    movel([0.094218, -1.402546, -2.554876, -0.754968, 1.570796, 1.665014],accel_mss,speed_ms,0,blend_radius_m)
    movel([0.093145, -1.402897, -2.554616, -0.754876, 1.570796, 1.663941],accel_mss,speed_ms,0,blend_radius_m)
    movel([0.092652, -1.403004, -2.554537, -0.754848, 1.570796, 1.663448],accel_mss,speed_ms,0,blend_radius_m)
    movel([0.092424, -1.402949, -2.554578, -0.754862, 1.570796, 1.663220],accel_mss,speed_ms,0,blend_radius_m)
    movel([0.092353, -1.402753, -2.554722, -0.754913, 1.570796, 1.663149],accel_mss,speed_ms,0,blend_radius_m)
    movel([0.092529, -1.402431, -2.554960, -0.754998, 1.570796, 1.663326],accel_mss,speed_ms,0,blend_radius_m)
    movel([0.093124, -1.402001, -2.555277, -0.755111, 1.570796, 1.663921],accel_mss,speed_ms,0,blend_radius_m)
    movel([0.094351, -1.401555, -2.555606, -0.755228, 1.570796, 1.665147],accel_mss,speed_ms,0,blend_radius_m)
    movel([0.095795, -1.401115, -2.555930, -0.755344, 1.570796, 1.666591],accel_mss,speed_ms,0,blend_radius_m)
    speed_ms = 0.003
    movel([0.095795, -1.404350, -2.557382, -0.750656, 1.570796, 1.666591],accel_mss,speed_ms,0,blend_radius_m)
    speed_ms = 0.007
    movel([0.097270, -1.403994, -2.557646, -0.750749, 1.570796, 1.668067],accel_mss,speed_ms,0,blend_radius_m)
    movel([0.098200, -1.403807, -2.557784, -0.750798, 1.570796, 1.668996],accel_mss,speed_ms,0,blend_radius_m)
    movel([0.098654, -1.403741, -2.557833, -0.750815, 1.570796, 1.669451],accel_mss,speed_ms,0,blend_radius_m)
    movel([0.098932, -1.403749, -2.557827, -0.750813, 1.570796, 1.669729],accel_mss,speed_ms,0,blend_radius_m)
    movel([0.099151, -1.403824, -2.557771, -0.750794, 1.570796, 1.669947],accel_mss,speed_ms,0,blend_radius_m)
    movel([0.099338, -1.403962, -2.557669, -0.750758, 1.570796, 1.670134],accel_mss,speed_ms,0,blend_radius_m)
    movel([0.099360, -1.404241, -2.557463, -0.750685, 1.570796, 1.670156],accel_mss,speed_ms,0,blend_radius_m)
    movel([0.099047, -1.404511, -2.557263, -0.750614, 1.570796, 1.669844],accel_mss,speed_ms,0,blend_radius_m)
    movel([0.098716, -1.404617, -2.557185, -0.750587, 1.570796, 1.669513],accel_mss,speed_ms,0,blend_radius_m)
    movel([0.098213, -1.404743, -2.557092, -0.750554, 1.570796, 1.669009],accel_mss,speed_ms,0,blend_radius_m)
    movel([0.097407, -1.404912, -2.556967, -0.750510, 1.570796, 1.668203],accel_mss,speed_ms,0,blend_radius_m)
    movel([0.096581, -1.405094, -2.556832, -0.750463, 1.570796, 1.667377],accel_mss,speed_ms,0,blend_radius_m)
    movel([0.095800, -1.405291, -2.556686, -0.750412, 1.570796, 1.666597],accel_mss,speed_ms,0,blend_radius_m)
    movel([0.095027, -1.405514, -2.556521, -0.750354, 1.570796, 1.665823],accel_mss,speed_ms,0,blend_radius_m)
    movel([0.094218, -1.405777, -2.556325, -0.750286, 1.570796, 1.665014],accel_mss,speed_ms,0,blend_radius_m)
    movel([0.093145, -1.406127, -2.556066, -0.750196, 1.570796, 1.663941],accel_mss,speed_ms,0,blend_radius_m)
    movel([0.092652, -1.406234, -2.555986, -0.750168, 1.570796, 1.663448],accel_mss,speed_ms,0,blend_radius_m)
    movel([0.092424, -1.406179, -2.556027, -0.750182, 1.570796, 1.663220],accel_mss,speed_ms,0,blend_radius_m)
    movel([0.092353, -1.405984, -2.556172, -0.750233, 1.570796, 1.663149],accel_mss,speed_ms,0,blend_radius_m)
    movel([0.092529, -1.405663, -2.556410, -0.750316, 1.570796, 1.663326],accel_mss,speed_ms,0,blend_radius_m)
    movel([0.093124, -1.405234, -2.556728, -0.750427, 1.570796, 1.663921],accel_mss,speed_ms,0,blend_radius_m)
    movel([0.094351, -1.404789, -2.557058, -0.750542, 1.570796, 1.665147],accel_mss,speed_ms,0,blend_radius_m)
    movel([0.095795, -1.404350, -2.557382, -0.750656, 1.570796, 1.666591],accel_mss,speed_ms,0,blend_radius_m)
    speed_ms = 0.003
    movel([0.095795, -1.391535, -2.551523, -0.769331, 1.570796, 1.666591],accel_mss,speed_ms,0,blend_radius_m)
    speed_ms = 1.000
    movel([0.095795, -1.366921, -2.539410, -0.806058, 1.570796, 1.666591],accel_mss,speed_ms,0,blend_radius_m)
    movel([0.095058, -1.368794, -2.538098, -0.805497, 1.570796, 1.665854],accel_mss,speed_ms,0,blend_radius_m)
    movel([0.095058, -1.393374, -2.550187, -0.768828, 1.570796, 1.665854],accel_mss,speed_ms,0,blend_radius_m)
    speed_ms = 0.003
    movel([0.095058, -1.402939, -2.554585, -0.754865, 1.570796, 1.665854],accel_mss,speed_ms,0,blend_radius_m)
    speed_ms = 0.007
    movel([0.096957, -1.402395, -2.554986, -0.755007, 1.570796, 1.667754],accel_mss,speed_ms,0,blend_radius_m)
    movel([0.098037, -1.402157, -2.555162, -0.755070, 1.570796, 1.668833],accel_mss,speed_ms,0,blend_radius_m)
    movel([0.098676, -1.402118, -2.555191, -0.755080, 1.570796, 1.669473],accel_mss,speed_ms,0,blend_radius_m)
    movel([0.099066, -1.402259, -2.555087, -0.755043, 1.570796, 1.669862],accel_mss,speed_ms,0,blend_radius_m)
    movel([0.099131, -1.402534, -2.554884, -0.754971, 1.570796, 1.669927],accel_mss,speed_ms,0,blend_radius_m)
    movel([0.098905, -1.402879, -2.554629, -0.754881, 1.570796, 1.669701],accel_mss,speed_ms,0,blend_radius_m)
    movel([0.098649, -1.402995, -2.554544, -0.754850, 1.570796, 1.669445],accel_mss,speed_ms,0,blend_radius_m)
    movel([0.098218, -1.403073, -2.554486, -0.754830, 1.570796, 1.669014],accel_mss,speed_ms,0,blend_radius_m)
    movel([0.097382, -1.403224, -2.554375, -0.754791, 1.570796, 1.668179],accel_mss,speed_ms,0,blend_radius_m)
    movel([0.095577, -1.403702, -2.554021, -0.754666, 1.570796, 1.666373],accel_mss,speed_ms,0,blend_radius_m)
    movel([0.093763, -1.404215, -2.553642, -0.754533, 1.570796, 1.664560],accel_mss,speed_ms,0,blend_radius_m)
    movel([0.092999, -1.404503, -2.553428, -0.754458, 1.570796, 1.663795],accel_mss,speed_ms,0,blend_radius_m)
    movel([0.092709, -1.404629, -2.553335, -0.754425, 1.570796, 1.663506],accel_mss,speed_ms,0,blend_radius_m)
    movel([0.092398, -1.404692, -2.553288, -0.754409, 1.570796, 1.663195],accel_mss,speed_ms,0,blend_radius_m)
    movel([0.092200, -1.404501, -2.553429, -0.754458, 1.570796, 1.662996],accel_mss,speed_ms,0,blend_radius_m)
    movel([0.092240, -1.404260, -2.553608, -0.754521, 1.570796, 1.663036],accel_mss,speed_ms,0,blend_radius_m)
    movel([0.092394, -1.403991, -2.553808, -0.754591, 1.570796, 1.663190],accel_mss,speed_ms,0,blend_radius_m)
    movel([0.092628, -1.403768, -2.553972, -0.754649, 1.570796, 1.663424],accel_mss,speed_ms,0,blend_radius_m)
    movel([0.093075, -1.403542, -2.554139, -0.754707, 1.570796, 1.663871],accel_mss,speed_ms,0,blend_radius_m)
    movel([0.095058, -1.402939, -2.554585, -0.754865, 1.570796, 1.665854],accel_mss,speed_ms,0,blend_radius_m)
    speed_ms = 0.003
    movel([0.095058, -1.406170, -2.556034, -0.750185, 1.570796, 1.665854],accel_mss,speed_ms,0,blend_radius_m)
    speed_ms = 0.007
    movel([0.096957, -1.405627, -2.556437, -0.750325, 1.570796, 1.667754],accel_mss,speed_ms,0,blend_radius_m)
    movel([0.098037, -1.405390, -2.556613, -0.750386, 1.570796, 1.668833],accel_mss,speed_ms,0,blend_radius_m)
    movel([0.098676, -1.405351, -2.556641, -0.750396, 1.570796, 1.669473],accel_mss,speed_ms,0,blend_radius_m)
    movel([0.099066, -1.405491, -2.556537, -0.750360, 1.570796, 1.669862],accel_mss,speed_ms,0,blend_radius_m)
    movel([0.099131, -1.405766, -2.556334, -0.750289, 1.570796, 1.669927],accel_mss,speed_ms,0,blend_radius_m)
    movel([0.098905, -1.406110, -2.556079, -0.750200, 1.570796, 1.669701],accel_mss,speed_ms,0,blend_radius_m)
    movel([0.098649, -1.406225, -2.555993, -0.750171, 1.570796, 1.669445],accel_mss,speed_ms,0,blend_radius_m)
    movel([0.098218, -1.406303, -2.555935, -0.750151, 1.570796, 1.669014],accel_mss,speed_ms,0,blend_radius_m)
    movel([0.097382, -1.406453, -2.555824, -0.750112, 1.570796, 1.668179],accel_mss,speed_ms,0,blend_radius_m)
    movel([0.095577, -1.406930, -2.555469, -0.749989, 1.570796, 1.666373],accel_mss,speed_ms,0,blend_radius_m)
    movel([0.093763, -1.407442, -2.555089, -0.749858, 1.570796, 1.664560],accel_mss,speed_ms,0,blend_radius_m)
    movel([0.092999, -1.407729, -2.554875, -0.749785, 1.570796, 1.663795],accel_mss,speed_ms,0,blend_radius_m)
    movel([0.092709, -1.407855, -2.554782, -0.749753, 1.570796, 1.663506],accel_mss,speed_ms,0,blend_radius_m)
    movel([0.092398, -1.407917, -2.554735, -0.749737, 1.570796, 1.663195],accel_mss,speed_ms,0,blend_radius_m)
    movel([0.092200, -1.407728, -2.554876, -0.749785, 1.570796, 1.662996],accel_mss,speed_ms,0,blend_radius_m)
    movel([0.092240, -1.407487, -2.555056, -0.749847, 1.570796, 1.663036],accel_mss,speed_ms,0,blend_radius_m)
    movel([0.092394, -1.407218, -2.555255, -0.749916, 1.570796, 1.663190],accel_mss,speed_ms,0,blend_radius_m)
    movel([0.092628, -1.406997, -2.555420, -0.749972, 1.570796, 1.663424],accel_mss,speed_ms,0,blend_radius_m)
    movel([0.093075, -1.406771, -2.555588, -0.750030, 1.570796, 1.663871],accel_mss,speed_ms,0,blend_radius_m)
    movel([0.095058, -1.406170, -2.556034, -0.750185, 1.570796, 1.665854],accel_mss,speed_ms,0,blend_radius_m)
    speed_ms = 0.003
    movel([0.095058, -1.393374, -2.550187, -0.768828, 1.570796, 1.665854],accel_mss,speed_ms,0,blend_radius_m)
    speed_ms = 1.000
    movel([0.095058, -1.368794, -2.538098, -0.805497, 1.570796, 1.665854],accel_mss,speed_ms,0,blend_radius_m)
    movel([0.095035, -1.370360, -2.536997, -0.805032, 1.570796, 1.665831],accel_mss,speed_ms,0,blend_radius_m)
    movel([0.095035, -1.394911, -2.549067, -0.768411, 1.570796, 1.665831],accel_mss,speed_ms,0,blend_radius_m)
    speed_ms = 0.003
    movel([0.095035, -1.404463, -2.553458, -0.754468, 1.570796, 1.665831],accel_mss,speed_ms,0,blend_radius_m)
    speed_ms = 0.007
    movel([0.096678, -1.404013, -2.553791, -0.754585, 1.570796, 1.667474],accel_mss,speed_ms,0,blend_radius_m)
    movel([0.097776, -1.403780, -2.553963, -0.754646, 1.570796, 1.668573],accel_mss,speed_ms,0,blend_radius_m)
    movel([0.098503, -1.403710, -2.554016, -0.754664, 1.570796, 1.669299],accel_mss,speed_ms,0,blend_radius_m)
    movel([0.098867, -1.403822, -2.553932, -0.754635, 1.570796, 1.669663],accel_mss,speed_ms,0,blend_radius_m)
    movel([0.098943, -1.404146, -2.553692, -0.754550, 1.570796, 1.669739],accel_mss,speed_ms,0,blend_radius_m)
    movel([0.098660, -1.404518, -2.553417, -0.754454, 1.570796, 1.669456],accel_mss,speed_ms,0,blend_radius_m)
    movel([0.098382, -1.404581, -2.553370, -0.754438, 1.570796, 1.669178],accel_mss,speed_ms,0,blend_radius_m)
    movel([0.098132, -1.404608, -2.553350, -0.754431, 1.570796, 1.668928],accel_mss,speed_ms,0,blend_radius_m)
    movel([0.097854, -1.404624, -2.553339, -0.754426, 1.570796, 1.668651],accel_mss,speed_ms,0,blend_radius_m)
    movel([0.096922, -1.404748, -2.553246, -0.754394, 1.570796, 1.667719],accel_mss,speed_ms,0,blend_radius_m)
    movel([0.095411, -1.405123, -2.552968, -0.754297, 1.570796, 1.666208],accel_mss,speed_ms,0,blend_radius_m)
    movel([0.093895, -1.405570, -2.552637, -0.754182, 1.570796, 1.664692],accel_mss,speed_ms,0,blend_radius_m)
    movel([0.092949, -1.405958, -2.552349, -0.754082, 1.570796, 1.663745],accel_mss,speed_ms,0,blend_radius_m)
    movel([0.092619, -1.406115, -2.552232, -0.754042, 1.570796, 1.663415],accel_mss,speed_ms,0,blend_radius_m)
    movel([0.092226, -1.406242, -2.552137, -0.754009, 1.570796, 1.663023],accel_mss,speed_ms,0,blend_radius_m)
    movel([0.092027, -1.406107, -2.552238, -0.754044, 1.570796, 1.662823],accel_mss,speed_ms,0,blend_radius_m)
    movel([0.092203, -1.405669, -2.552563, -0.754157, 1.570796, 1.663000],accel_mss,speed_ms,0,blend_radius_m)
    movel([0.092457, -1.405414, -2.552753, -0.754222, 1.570796, 1.663253],accel_mss,speed_ms,0,blend_radius_m)
    movel([0.092744, -1.405218, -2.552898, -0.754273, 1.570796, 1.663541],accel_mss,speed_ms,0,blend_radius_m)
    movel([0.093114, -1.405050, -2.553023, -0.754316, 1.570796, 1.663910],accel_mss,speed_ms,0,blend_radius_m)
    movel([0.093718, -1.404848, -2.553172, -0.754368, 1.570796, 1.664514],accel_mss,speed_ms,0,blend_radius_m)
    movel([0.095035, -1.404463, -2.553458, -0.754468, 1.570796, 1.665831],accel_mss,speed_ms,0,blend_radius_m)
    speed_ms = 0.003
    movel([0.095035, -1.407689, -2.554905, -0.749795, 1.570796, 1.665831],accel_mss,speed_ms,0,blend_radius_m)
    speed_ms = 0.007
    movel([0.096678, -1.407240, -2.555239, -0.749910, 1.570796, 1.667474],accel_mss,speed_ms,0,blend_radius_m)
    movel([0.097776, -1.407008, -2.555411, -0.749969, 1.570796, 1.668573],accel_mss,speed_ms,0,blend_radius_m)
    movel([0.098503, -1.406938, -2.555464, -0.749987, 1.570796, 1.669299],accel_mss,speed_ms,0,blend_radius_m)
    movel([0.098867, -1.407050, -2.555380, -0.749959, 1.570796, 1.669663],accel_mss,speed_ms,0,blend_radius_m)
    movel([0.098943, -1.407374, -2.555140, -0.749876, 1.570796, 1.669739],accel_mss,speed_ms,0,blend_radius_m)
    movel([0.098660, -1.407744, -2.554864, -0.749781, 1.570796, 1.669456],accel_mss,speed_ms,0,blend_radius_m)
    movel([0.098382, -1.407807, -2.554817, -0.749765, 1.570796, 1.669178],accel_mss,speed_ms,0,blend_radius_m)
    movel([0.098132, -1.407834, -2.554797, -0.749758, 1.570796, 1.668928],accel_mss,speed_ms,0,blend_radius_m)
    movel([0.097854, -1.407850, -2.554785, -0.749754, 1.570796, 1.668651],accel_mss,speed_ms,0,blend_radius_m)
    movel([0.096922, -1.407974, -2.554693, -0.749722, 1.570796, 1.667719],accel_mss,speed_ms,0,blend_radius_m)
    movel([0.095411, -1.408348, -2.554414, -0.749627, 1.570796, 1.666208],accel_mss,speed_ms,0,blend_radius_m)
    movel([0.093895, -1.408794, -2.554082, -0.749514, 1.570796, 1.664692],accel_mss,speed_ms,0,blend_radius_m)
    movel([0.092949, -1.409180, -2.553793, -0.749416, 1.570796, 1.663745],accel_mss,speed_ms,0,blend_radius_m)
    movel([0.092619, -1.409336, -2.553676, -0.749376, 1.570796, 1.663415],accel_mss,speed_ms,0,blend_radius_m)
    movel([0.092226, -1.409464, -2.553581, -0.749344, 1.570796, 1.663023],accel_mss,speed_ms,0,blend_radius_m)
    movel([0.092027, -1.409329, -2.553682, -0.749378, 1.570796, 1.662823],accel_mss,speed_ms,0,blend_radius_m)
    movel([0.092203, -1.408892, -2.554008, -0.749489, 1.570796, 1.663000],accel_mss,speed_ms,0,blend_radius_m)
    movel([0.092457, -1.408637, -2.554198, -0.749553, 1.570796, 1.663253],accel_mss,speed_ms,0,blend_radius_m)
    movel([0.092744, -1.408442, -2.554344, -0.749603, 1.570796, 1.663541],accel_mss,speed_ms,0,blend_radius_m)
    movel([0.093114, -1.408275, -2.554469, -0.749646, 1.570796, 1.663910],accel_mss,speed_ms,0,blend_radius_m)
    movel([0.093718, -1.408074, -2.554618, -0.749697, 1.570796, 1.664514],accel_mss,speed_ms,0,blend_radius_m)
    movel([0.095035, -1.407689, -2.554905, -0.749795, 1.570796, 1.665831],accel_mss,speed_ms,0,blend_radius_m)
    speed_ms = 0.003
    movel([0.095035, -1.394911, -2.549067, -0.768411, 1.570796, 1.665831],accel_mss,speed_ms,0,blend_radius_m)
    speed_ms = 1.000
    movel([0.095035, -1.370360, -2.536997, -0.805032, 1.570796, 1.665831],accel_mss,speed_ms,0,blend_radius_m)
    movel([0.094639, -1.371914, -2.535902, -0.804573, 1.570796, 1.665435],accel_mss,speed_ms,0,blend_radius_m)
    movel([0.094639, -1.396436, -2.547952, -0.768001, 1.570796, 1.665435],accel_mss,speed_ms,0,blend_radius_m)
    speed_ms = 0.003
    movel([0.094639, -1.405976, -2.552335, -0.754078, 1.570796, 1.665435],accel_mss,speed_ms,0,blend_radius_m)
    speed_ms = 0.007
    movel([0.095700, -1.405698, -2.552542, -0.754149, 1.570796, 1.666496],accel_mss,speed_ms,0,blend_radius_m)
    movel([0.097708, -1.405190, -2.552919, -0.754280, 1.570796, 1.668504],accel_mss,speed_ms,0,blend_radius_m)
    movel([0.098496, -1.405331, -2.552814, -0.754244, 1.570796, 1.669292],accel_mss,speed_ms,0,blend_radius_m)
    movel([0.099084, -1.405493, -2.552694, -0.754202, 1.570796, 1.669880],accel_mss,speed_ms,0,blend_radius_m)
    movel([0.099446, -1.405731, -2.552517, -0.754141, 1.570796, 1.670242],accel_mss,speed_ms,0,blend_radius_m)
    movel([0.099663, -1.406106, -2.552239, -0.754044, 1.570796, 1.670460],accel_mss,speed_ms,0,blend_radius_m)
    movel([0.099786, -1.406703, -2.551795, -0.753891, 1.570796, 1.670583],accel_mss,speed_ms,0,blend_radius_m)
    movel([0.099688, -1.407004, -2.551571, -0.753814, 1.570796, 1.670484],accel_mss,speed_ms,0,blend_radius_m)
    movel([0.099544, -1.407333, -2.551326, -0.753730, 1.570796, 1.670341],accel_mss,speed_ms,0,blend_radius_m)
    movel([0.099344, -1.407622, -2.551110, -0.753657, 1.570796, 1.670140],accel_mss,speed_ms,0,blend_radius_m)
    movel([0.098360, -1.408089, -2.550762, -0.753538, 1.570796, 1.669156],accel_mss,speed_ms,0,blend_radius_m)
    movel([0.096049, -1.408788, -2.550240, -0.753361, 1.570796, 1.666845],accel_mss,speed_ms,0,blend_radius_m)
    movel([0.093670, -1.409447, -2.549747, -0.753195, 1.570796, 1.664466],accel_mss,speed_ms,0,blend_radius_m)
    movel([0.091851, -1.409859, -2.549439, -0.753091, 1.570796, 1.662647],accel_mss,speed_ms,0,blend_radius_m)
    movel([0.091060, -1.409980, -2.549348, -0.753061, 1.570796, 1.661856],accel_mss,speed_ms,0,blend_radius_m)
    movel([0.090671, -1.409936, -2.549381, -0.753072, 1.570796, 1.661467],accel_mss,speed_ms,0,blend_radius_m)
    movel([0.090493, -1.409731, -2.549535, -0.753123, 1.570796, 1.661289],accel_mss,speed_ms,0,blend_radius_m)
    movel([0.090475, -1.409302, -2.549856, -0.753231, 1.570796, 1.661272],accel_mss,speed_ms,0,blend_radius_m)
    movel([0.090698, -1.408553, -2.550415, -0.753420, 1.570796, 1.661494],accel_mss,speed_ms,0,blend_radius_m)
    movel([0.091185, -1.407836, -2.550951, -0.753602, 1.570796, 1.661982],accel_mss,speed_ms,0,blend_radius_m)
    movel([0.091933, -1.407176, -2.551443, -0.753770, 1.570796, 1.662729],accel_mss,speed_ms,0,blend_radius_m)
    movel([0.092913, -1.406594, -2.551876, -0.753919, 1.570796, 1.663709],accel_mss,speed_ms,0,blend_radius_m)
    movel([0.093405, -1.406375, -2.552039, -0.753975, 1.570796, 1.664201],accel_mss,speed_ms,0,blend_radius_m)
    movel([0.093939, -1.406183, -2.552182, -0.754025, 1.570796, 1.664735],accel_mss,speed_ms,0,blend_radius_m)
    movel([0.094639, -1.405976, -2.552335, -0.754078, 1.570796, 1.665435],accel_mss,speed_ms,0,blend_radius_m)
    speed_ms = 0.003
    movel([0.094639, -1.409198, -2.553780, -0.749411, 1.570796, 1.665435],accel_mss,speed_ms,0,blend_radius_m)
    speed_ms = 0.007
    movel([0.095700, -1.408921, -2.553987, -0.749481, 1.570796, 1.666496],accel_mss,speed_ms,0,blend_radius_m)
    movel([0.097708, -1.408414, -2.554365, -0.749610, 1.570796, 1.668504],accel_mss,speed_ms,0,blend_radius_m)
    movel([0.098496, -1.408555, -2.554259, -0.749574, 1.570796, 1.669292],accel_mss,speed_ms,0,blend_radius_m)
    movel([0.099084, -1.408716, -2.554139, -0.749533, 1.570796, 1.669880],accel_mss,speed_ms,0,blend_radius_m)
    movel([0.099446, -1.408954, -2.553962, -0.749473, 1.570796, 1.670242],accel_mss,speed_ms,0,blend_radius_m)
    movel([0.099663, -1.409327, -2.553683, -0.749379, 1.570796, 1.670460],accel_mss,speed_ms,0,blend_radius_m)
    movel([0.099786, -1.409923, -2.553238, -0.749228, 1.570796, 1.670583],accel_mss,speed_ms,0,blend_radius_m)
    movel([0.099688, -1.410223, -2.553014, -0.749152, 1.570796, 1.670484],accel_mss,speed_ms,0,blend_radius_m)
    movel([0.099544, -1.410551, -2.552768, -0.749070, 1.570796, 1.670341],accel_mss,speed_ms,0,blend_radius_m)
    movel([0.099344, -1.410840, -2.552552, -0.748998, 1.570796, 1.670140],accel_mss,speed_ms,0,blend_radius_m)
    movel([0.098360, -1.411305, -2.552203, -0.748881, 1.570796, 1.669156],accel_mss,speed_ms,0,blend_radius_m)
    movel([0.096049, -1.412002, -2.551680, -0.748707, 1.570796, 1.666845],accel_mss,speed_ms,0,blend_radius_m)
    movel([0.093670, -1.412659, -2.551186, -0.748544, 1.570796, 1.664466],accel_mss,speed_ms,0,blend_radius_m)
    movel([0.091851, -1.413070, -2.550877, -0.748442, 1.570796, 1.662647],accel_mss,speed_ms,0,blend_radius_m)
    movel([0.091060, -1.413191, -2.550786, -0.748412, 1.570796, 1.661856],accel_mss,speed_ms,0,blend_radius_m)
    movel([0.090671, -1.413147, -2.550820, -0.748423, 1.570796, 1.661467],accel_mss,speed_ms,0,blend_radius_m)
    movel([0.090493, -1.412943, -2.550973, -0.748473, 1.570796, 1.661289],accel_mss,speed_ms,0,blend_radius_m)
    movel([0.090475, -1.412515, -2.551295, -0.748579, 1.570796, 1.661272],accel_mss,speed_ms,0,blend_radius_m)
    movel([0.090698, -1.411768, -2.551856, -0.748765, 1.570796, 1.661494],accel_mss,speed_ms,0,blend_radius_m)
    movel([0.091185, -1.411053, -2.552392, -0.748944, 1.570796, 1.661982],accel_mss,speed_ms,0,blend_radius_m)
    movel([0.091933, -1.410395, -2.552885, -0.749109, 1.570796, 1.662729],accel_mss,speed_ms,0,blend_radius_m)
    movel([0.092913, -1.409814, -2.553319, -0.749256, 1.570796, 1.663709],accel_mss,speed_ms,0,blend_radius_m)
    movel([0.093405, -1.409596, -2.553483, -0.749311, 1.570796, 1.664201],accel_mss,speed_ms,0,blend_radius_m)
    movel([0.093939, -1.409404, -2.553626, -0.749359, 1.570796, 1.664735],accel_mss,speed_ms,0,blend_radius_m)
    movel([0.094639, -1.409198, -2.553780, -0.749411, 1.570796, 1.665435],accel_mss,speed_ms,0,blend_radius_m)
    speed_ms = 0.003
    movel([0.094639, -1.396436, -2.547952, -0.768001, 1.570796, 1.665435],accel_mss,speed_ms,0,blend_radius_m)
    speed_ms = 1.000
    movel([0.094639, -1.371914, -2.535902, -0.804573, 1.570796, 1.665435],accel_mss,speed_ms,0,blend_radius_m)
    movel([0.105149, -1.357142, -2.546182, -0.809066, 1.570796, 1.675945],accel_mss,speed_ms,0,blend_radius_m)
    movel([0.105149, -1.381936, -2.558418, -0.772035, 1.570796, 1.675945],accel_mss,speed_ms,0,blend_radius_m)
    speed_ms = 0.003
    movel([0.105149, -1.391592, -2.562871, -0.757926, 1.570796, 1.675945],accel_mss,speed_ms,0,blend_radius_m)
    speed_ms = 0.007
    movel([0.104563, -1.391094, -2.563231, -0.758064, 1.570796, 1.675360],accel_mss,speed_ms,0,blend_radius_m)
    movel([0.104458, -1.390234, -2.563850, -0.758305, 1.570796, 1.675254],accel_mss,speed_ms,0,blend_radius_m)
    movel([0.104866, -1.389249, -2.564559, -0.758581, 1.570796, 1.675663],accel_mss,speed_ms,0,blend_radius_m)
    movel([0.105135, -1.388888, -2.564818, -0.758683, 1.570796, 1.675931],accel_mss,speed_ms,0,blend_radius_m)
    movel([0.105367, -1.388728, -2.564933, -0.758728, 1.570796, 1.676164],accel_mss,speed_ms,0,blend_radius_m)
    movel([0.105422, -1.389121, -2.564651, -0.758617, 1.570796, 1.676219],accel_mss,speed_ms,0,blend_radius_m)
    movel([0.105424, -1.389397, -2.564452, -0.758539, 1.570796, 1.676221],accel_mss,speed_ms,0,blend_radius_m)
    movel([0.105462, -1.390010, -2.564012, -0.758367, 1.570796, 1.676258],accel_mss,speed_ms,0,blend_radius_m)
    movel([0.105618, -1.390484, -2.563670, -0.758235, 1.570796, 1.676415],accel_mss,speed_ms,0,blend_radius_m)
    movel([0.105896, -1.390824, -2.563425, -0.758140, 1.570796, 1.676693],accel_mss,speed_ms,0,blend_radius_m)
    movel([0.106295, -1.391039, -2.563270, -0.758080, 1.570796, 1.677091],accel_mss,speed_ms,0,blend_radius_m)
    movel([0.106601, -1.391184, -2.563166, -0.758039, 1.570796, 1.677397],accel_mss,speed_ms,0,blend_radius_m)
    movel([0.106634, -1.391377, -2.563026, -0.757985, 1.570796, 1.677431],accel_mss,speed_ms,0,blend_radius_m)
    movel([0.106282, -1.391530, -2.562916, -0.757943, 1.570796, 1.677078],accel_mss,speed_ms,0,blend_radius_m)
    movel([0.105149, -1.391592, -2.562871, -0.757926, 1.570796, 1.675945],accel_mss,speed_ms,0,blend_radius_m)
    speed_ms = 0.003
    movel([0.105149, -1.394854, -2.564339, -0.753196, 1.570796, 1.675945],accel_mss,speed_ms,0,blend_radius_m)
    speed_ms = 0.007
    movel([0.104563, -1.394357, -2.564699, -0.753332, 1.570796, 1.675360],accel_mss,speed_ms,0,blend_radius_m)
    movel([0.104458, -1.393500, -2.565320, -0.753569, 1.570796, 1.675254],accel_mss,speed_ms,0,blend_radius_m)
    movel([0.104866, -1.392517, -2.566031, -0.753841, 1.570796, 1.675663],accel_mss,speed_ms,0,blend_radius_m)
    movel([0.105135, -1.392158, -2.566290, -0.753941, 1.570796, 1.675931],accel_mss,speed_ms,0,blend_radius_m)
    movel([0.105367, -1.391998, -2.566406, -0.753986, 1.570796, 1.676164],accel_mss,speed_ms,0,blend_radius_m)
    movel([0.105422, -1.392390, -2.566123, -0.753877, 1.570796, 1.676219],accel_mss,speed_ms,0,blend_radius_m)
    movel([0.105424, -1.392666, -2.565923, -0.753800, 1.570796, 1.676221],accel_mss,speed_ms,0,blend_radius_m)
    movel([0.105462, -1.393277, -2.565482, -0.753631, 1.570796, 1.676258],accel_mss,speed_ms,0,blend_radius_m)
    movel([0.105618, -1.393750, -2.565140, -0.753500, 1.570796, 1.676415],accel_mss,speed_ms,0,blend_radius_m)
    movel([0.105896, -1.394089, -2.564894, -0.753406, 1.570796, 1.676693],accel_mss,speed_ms,0,blend_radius_m)
    movel([0.106295, -1.394303, -2.564739, -0.753347, 1.570796, 1.677091],accel_mss,speed_ms,0,blend_radius_m)
    movel([0.106601, -1.394447, -2.564634, -0.753308, 1.570796, 1.677397],accel_mss,speed_ms,0,blend_radius_m)
    movel([0.106634, -1.394640, -2.564494, -0.753255, 1.570796, 1.677431],accel_mss,speed_ms,0,blend_radius_m)
    movel([0.106282, -1.394792, -2.564384, -0.753213, 1.570796, 1.677078],accel_mss,speed_ms,0,blend_radius_m)
    movel([0.105149, -1.394854, -2.564339, -0.753196, 1.570796, 1.675945],accel_mss,speed_ms,0,blend_radius_m)
    speed_ms = 0.003
    movel([0.105149, -1.381936, -2.558418, -0.772035, 1.570796, 1.675945],accel_mss,speed_ms,0,blend_radius_m)
    speed_ms = 1.000
    movel([0.105149, -1.357142, -2.546182, -0.809066, 1.570796, 1.675945],accel_mss,speed_ms,0,blend_radius_m)
    movel([0.110232, -1.354325, -2.548108, -0.809956, 1.570796, 1.681029],accel_mss,speed_ms,0,blend_radius_m)
    movel([0.110232, -1.379170, -2.560380, -0.772838, 1.570796, 1.681029],accel_mss,speed_ms,0,blend_radius_m)
    speed_ms = 0.003
    movel([0.110232, -1.388848, -2.564847, -0.758694, 1.570796, 1.681029],accel_mss,speed_ms,0,blend_radius_m)
    speed_ms = 0.007
    movel([0.110305, -1.388373, -2.565188, -0.758828, 1.570796, 1.681101],accel_mss,speed_ms,0,blend_radius_m)
    movel([0.110347, -1.387801, -2.565598, -0.758990, 1.570796, 1.681143],accel_mss,speed_ms,0,blend_radius_m)
    movel([0.110245, -1.387322, -2.565941, -0.759126, 1.570796, 1.681042],accel_mss,speed_ms,0,blend_radius_m)
    movel([0.109999, -1.386943, -2.566212, -0.759234, 1.570796, 1.680796],accel_mss,speed_ms,0,blend_radius_m)
    movel([0.109609, -1.386664, -2.566412, -0.759314, 1.570796, 1.680405],accel_mss,speed_ms,0,blend_radius_m)
    movel([0.109341, -1.386511, -2.566521, -0.759357, 1.570796, 1.680137],accel_mss,speed_ms,0,blend_radius_m)
    movel([0.109697, -1.386266, -2.566696, -0.759427, 1.570796, 1.680494],accel_mss,speed_ms,0,blend_radius_m)
    movel([0.110064, -1.386321, -2.566656, -0.759411, 1.570796, 1.680860],accel_mss,speed_ms,0,blend_radius_m)
    movel([0.110479, -1.386543, -2.566498, -0.759348, 1.570796, 1.681275],accel_mss,speed_ms,0,blend_radius_m)
    movel([0.110833, -1.386845, -2.566282, -0.759262, 1.570796, 1.681629],accel_mss,speed_ms,0,blend_radius_m)
    movel([0.111019, -1.387167, -2.566052, -0.759170, 1.570796, 1.681815],accel_mss,speed_ms,0,blend_radius_m)
    movel([0.111077, -1.387536, -2.565788, -0.759065, 1.570796, 1.681873],accel_mss,speed_ms,0,blend_radius_m)
    movel([0.111027, -1.387962, -2.565482, -0.758945, 1.570796, 1.681823],accel_mss,speed_ms,0,blend_radius_m)
    movel([0.110881, -1.388389, -2.565176, -0.758824, 1.570796, 1.681677],accel_mss,speed_ms,0,blend_radius_m)
    movel([0.110658, -1.388753, -2.564915, -0.758721, 1.570796, 1.681454],accel_mss,speed_ms,0,blend_radius_m)
    movel([0.110420, -1.389003, -2.564736, -0.758650, 1.570796, 1.681217],accel_mss,speed_ms,0,blend_radius_m)
    movel([0.110232, -1.388848, -2.564847, -0.758694, 1.570796, 1.681029],accel_mss,speed_ms,0,blend_radius_m)
    speed_ms = 0.003
    movel([0.110232, -1.392118, -2.566319, -0.753952, 1.570796, 1.681029],accel_mss,speed_ms,0,blend_radius_m)
    speed_ms = 0.007
    movel([0.110305, -1.391644, -2.566661, -0.754084, 1.570796, 1.681101],accel_mss,speed_ms,0,blend_radius_m)
    movel([0.110347, -1.391074, -2.567071, -0.754244, 1.570796, 1.681143],accel_mss,speed_ms,0,blend_radius_m)
    movel([0.110245, -1.390596, -2.567416, -0.754378, 1.570796, 1.681042],accel_mss,speed_ms,0,blend_radius_m)
    movel([0.109999, -1.390218, -2.567687, -0.754484, 1.570796, 1.680796],accel_mss,speed_ms,0,blend_radius_m)
    movel([0.109609, -1.389940, -2.567887, -0.754562, 1.570796, 1.680405],accel_mss,speed_ms,0,blend_radius_m)
    movel([0.109341, -1.389788, -2.567997, -0.754605, 1.570796, 1.680137],accel_mss,speed_ms,0,blend_radius_m)
    movel([0.109697, -1.389543, -2.568172, -0.754674, 1.570796, 1.680494],accel_mss,speed_ms,0,blend_radius_m)
    movel([0.110064, -1.389598, -2.568133, -0.754658, 1.570796, 1.680860],accel_mss,speed_ms,0,blend_radius_m)
    movel([0.110479, -1.389819, -2.567974, -0.754596, 1.570796, 1.681275],accel_mss,speed_ms,0,blend_radius_m)
    movel([0.110833, -1.390120, -2.567758, -0.754511, 1.570796, 1.681629],accel_mss,speed_ms,0,blend_radius_m)
    movel([0.111019, -1.390441, -2.567527, -0.754421, 1.570796, 1.681815],accel_mss,speed_ms,0,blend_radius_m)
    movel([0.111077, -1.390809, -2.567262, -0.754318, 1.570796, 1.681873],accel_mss,speed_ms,0,blend_radius_m)
    movel([0.111027, -1.391234, -2.566956, -0.754199, 1.570796, 1.681823],accel_mss,speed_ms,0,blend_radius_m)
    movel([0.110881, -1.391660, -2.566649, -0.754080, 1.570796, 1.681677],accel_mss,speed_ms,0,blend_radius_m)
    movel([0.110658, -1.392023, -2.566387, -0.753979, 1.570796, 1.681454],accel_mss,speed_ms,0,blend_radius_m)
    movel([0.110420, -1.392272, -2.566208, -0.753909, 1.570796, 1.681217],accel_mss,speed_ms,0,blend_radius_m)
    movel([0.110232, -1.392118, -2.566319, -0.753952, 1.570796, 1.681029],accel_mss,speed_ms,0,blend_radius_m)
    speed_ms = 0.003
    movel([0.110232, -1.379170, -2.560380, -0.772838, 1.570796, 1.681029],accel_mss,speed_ms,0,blend_radius_m)
    speed_ms = 1.000
    movel([0.110232, -1.354325, -2.548108, -0.809956, 1.570796, 1.681029],accel_mss,speed_ms,0,blend_radius_m)
    movel([0.107803, -1.351830, -2.549806, -0.810754, 1.570796, 1.678599],accel_mss,speed_ms,0,blend_radius_m)
    movel([0.107803, -1.376720, -2.562109, -0.773559, 1.570796, 1.678599],accel_mss,speed_ms,0,blend_radius_m)
    speed_ms = 0.003
    movel([0.107803, -1.386417, -2.566588, -0.759384, 1.570796, 1.678599],accel_mss,speed_ms,0,blend_radius_m)
    speed_ms = 0.007
    movel([0.107128, -1.386811, -2.566306, -0.759272, 1.570796, 1.677924],accel_mss,speed_ms,0,blend_radius_m)
    movel([0.106731, -1.386981, -2.566185, -0.759223, 1.570796, 1.677527],accel_mss,speed_ms,0,blend_radius_m)
    movel([0.106421, -1.387067, -2.566123, -0.759199, 1.570796, 1.677217],accel_mss,speed_ms,0,blend_radius_m)
    movel([0.106109, -1.386952, -2.566205, -0.759231, 1.570796, 1.676905],accel_mss,speed_ms,0,blend_radius_m)
    movel([0.106253, -1.386718, -2.566373, -0.759298, 1.570796, 1.677049],accel_mss,speed_ms,0,blend_radius_m)
    movel([0.106611, -1.386494, -2.566533, -0.759362, 1.570796, 1.677408],accel_mss,speed_ms,0,blend_radius_m)
    movel([0.107012, -1.386281, -2.566685, -0.759423, 1.570796, 1.677808],accel_mss,speed_ms,0,blend_radius_m)
    movel([0.107410, -1.386119, -2.566801, -0.759469, 1.570796, 1.678207],accel_mss,speed_ms,0,blend_radius_m)
    movel([0.107741, -1.386026, -2.566867, -0.759496, 1.570796, 1.678537],accel_mss,speed_ms,0,blend_radius_m)
    movel([0.107964, -1.386144, -2.566783, -0.759462, 1.570796, 1.678760],accel_mss,speed_ms,0,blend_radius_m)
    movel([0.107803, -1.386417, -2.566588, -0.759384, 1.570796, 1.678599],accel_mss,speed_ms,0,blend_radius_m)
    speed_ms = 0.003
    movel([0.107803, -1.389693, -2.568064, -0.754631, 1.570796, 1.678599],accel_mss,speed_ms,0,blend_radius_m)
    speed_ms = 0.007
    movel([0.107128, -1.390086, -2.567782, -0.754521, 1.570796, 1.677924],accel_mss,speed_ms,0,blend_radius_m)
    movel([0.106731, -1.390256, -2.567660, -0.754473, 1.570796, 1.677527],accel_mss,speed_ms,0,blend_radius_m)
    movel([0.106421, -1.390342, -2.567598, -0.754449, 1.570796, 1.677217],accel_mss,speed_ms,0,blend_radius_m)
    movel([0.106109, -1.390227, -2.567681, -0.754481, 1.570796, 1.676905],accel_mss,speed_ms,0,blend_radius_m)
    movel([0.106253, -1.389994, -2.567849, -0.754547, 1.570796, 1.677049],accel_mss,speed_ms,0,blend_radius_m)
    movel([0.106611, -1.389770, -2.568009, -0.754610, 1.570796, 1.677408],accel_mss,speed_ms,0,blend_radius_m)
    movel([0.107012, -1.389558, -2.568161, -0.754669, 1.570796, 1.677808],accel_mss,speed_ms,0,blend_radius_m)
    movel([0.107410, -1.389397, -2.568277, -0.754715, 1.570796, 1.678207],accel_mss,speed_ms,0,blend_radius_m)
    movel([0.107741, -1.389303, -2.568344, -0.754741, 1.570796, 1.678537],accel_mss,speed_ms,0,blend_radius_m)
    movel([0.107964, -1.389422, -2.568259, -0.754708, 1.570796, 1.678760],accel_mss,speed_ms,0,blend_radius_m)
    movel([0.107803, -1.389693, -2.568064, -0.754631, 1.570796, 1.678599],accel_mss,speed_ms,0,blend_radius_m)
    speed_ms = 0.003
    movel([0.107803, -1.376720, -2.562109, -0.773559, 1.570796, 1.678599],accel_mss,speed_ms,0,blend_radius_m)
    speed_ms = 1.000
    movel([0.107803, -1.351830, -2.549806, -0.810754, 1.570796, 1.678599],accel_mss,speed_ms,0,blend_radius_m)
    movel([0.107973, -1.350503, -2.550705, -0.811181, 1.570796, 1.678770],accel_mss,speed_ms,0,blend_radius_m)
    movel([0.107973, -1.375417, -2.563025, -0.773946, 1.570796, 1.678770],accel_mss,speed_ms,0,blend_radius_m)
    speed_ms = 0.003
    movel([0.107973, -1.385124, -2.567510, -0.759754, 1.570796, 1.678770],accel_mss,speed_ms,0,blend_radius_m)
    speed_ms = 0.007
    movel([0.107603, -1.385250, -2.567421, -0.759718, 1.570796, 1.678399],accel_mss,speed_ms,0,blend_radius_m)
    movel([0.107189, -1.385395, -2.567317, -0.759676, 1.570796, 1.677985],accel_mss,speed_ms,0,blend_radius_m)
    movel([0.106724, -1.385579, -2.567186, -0.759624, 1.570796, 1.677521],accel_mss,speed_ms,0,blend_radius_m)
    movel([0.106276, -1.385774, -2.567047, -0.759568, 1.570796, 1.677072],accel_mss,speed_ms,0,blend_radius_m)
    movel([0.105926, -1.385946, -2.566924, -0.759519, 1.570796, 1.676722],accel_mss,speed_ms,0,blend_radius_m)
    movel([0.105544, -1.386142, -2.566785, -0.759463, 1.570796, 1.676341],accel_mss,speed_ms,0,blend_radius_m)
    movel([0.105157, -1.386272, -2.566691, -0.759425, 1.570796, 1.675953],accel_mss,speed_ms,0,blend_radius_m)
    movel([0.105004, -1.386071, -2.566835, -0.759483, 1.570796, 1.675800],accel_mss,speed_ms,0,blend_radius_m)
    movel([0.105156, -1.385786, -2.567039, -0.759564, 1.570796, 1.675952],accel_mss,speed_ms,0,blend_radius_m)
    movel([0.105471, -1.385463, -2.567269, -0.759657, 1.570796, 1.676268],accel_mss,speed_ms,0,blend_radius_m)
    movel([0.105874, -1.385190, -2.567463, -0.759735, 1.570796, 1.676671],accel_mss,speed_ms,0,blend_radius_m)
    movel([0.106140, -1.385062, -2.567555, -0.759772, 1.570796, 1.676936],accel_mss,speed_ms,0,blend_radius_m)
    movel([0.106547, -1.384893, -2.567675, -0.759821, 1.570796, 1.677344],accel_mss,speed_ms,0,blend_radius_m)
    movel([0.107006, -1.384720, -2.567798, -0.759871, 1.570796, 1.677802],accel_mss,speed_ms,0,blend_radius_m)
    movel([0.107455, -1.384567, -2.567907, -0.759915, 1.570796, 1.678251],accel_mss,speed_ms,0,blend_radius_m)
    movel([0.108037, -1.384386, -2.568036, -0.759967, 1.570796, 1.678833],accel_mss,speed_ms,0,blend_radius_m)
    movel([0.108361, -1.384309, -2.568091, -0.759989, 1.570796, 1.679158],accel_mss,speed_ms,0,blend_radius_m)
    movel([0.108712, -1.384347, -2.568064, -0.759978, 1.570796, 1.679508],accel_mss,speed_ms,0,blend_radius_m)
    movel([0.108880, -1.384554, -2.567917, -0.759918, 1.570796, 1.679677],accel_mss,speed_ms,0,blend_radius_m)
    movel([0.108710, -1.384798, -2.567743, -0.759848, 1.570796, 1.679507],accel_mss,speed_ms,0,blend_radius_m)
    movel([0.108314, -1.384993, -2.567604, -0.759792, 1.570796, 1.679110],accel_mss,speed_ms,0,blend_radius_m)
    movel([0.107973, -1.385124, -2.567510, -0.759754, 1.570796, 1.678770],accel_mss,speed_ms,0,blend_radius_m)
    speed_ms = 0.003
    movel([0.107973, -1.388404, -2.568989, -0.754996, 1.570796, 1.678770],accel_mss,speed_ms,0,blend_radius_m)
    speed_ms = 0.007
    movel([0.107603, -1.388529, -2.568899, -0.754961, 1.570796, 1.678399],accel_mss,speed_ms,0,blend_radius_m)
    movel([0.107189, -1.388675, -2.568795, -0.754919, 1.570796, 1.677985],accel_mss,speed_ms,0,blend_radius_m)
    movel([0.106724, -1.388858, -2.568663, -0.754867, 1.570796, 1.677521],accel_mss,speed_ms,0,blend_radius_m)
    movel([0.106276, -1.389052, -2.568524, -0.754812, 1.570796, 1.677072],accel_mss,speed_ms,0,blend_radius_m)
    movel([0.105926, -1.389224, -2.568401, -0.754764, 1.570796, 1.676722],accel_mss,speed_ms,0,blend_radius_m)
    movel([0.105544, -1.389419, -2.568261, -0.754709, 1.570796, 1.676341],accel_mss,speed_ms,0,blend_radius_m)
    movel([0.105157, -1.389549, -2.568168, -0.754672, 1.570796, 1.675953],accel_mss,speed_ms,0,blend_radius_m)
    movel([0.105004, -1.389348, -2.568312, -0.754729, 1.570796, 1.675800],accel_mss,speed_ms,0,blend_radius_m)
    movel([0.105156, -1.389064, -2.568516, -0.754809, 1.570796, 1.675952],accel_mss,speed_ms,0,blend_radius_m)
    movel([0.105471, -1.388742, -2.568747, -0.754900, 1.570796, 1.676268],accel_mss,speed_ms,0,blend_radius_m)
    movel([0.105874, -1.388470, -2.568941, -0.754977, 1.570796, 1.676671],accel_mss,speed_ms,0,blend_radius_m)
    movel([0.106140, -1.388342, -2.569033, -0.755014, 1.570796, 1.676936],accel_mss,speed_ms,0,blend_radius_m)
    movel([0.106547, -1.388173, -2.569154, -0.755062, 1.570796, 1.677344],accel_mss,speed_ms,0,blend_radius_m)
    movel([0.107006, -1.388001, -2.569277, -0.755111, 1.570796, 1.677802],accel_mss,speed_ms,0,blend_radius_m)
    movel([0.107455, -1.387849, -2.569386, -0.755154, 1.570796, 1.678251],accel_mss,speed_ms,0,blend_radius_m)
    movel([0.108037, -1.387668, -2.569515, -0.755205, 1.570796, 1.678833],accel_mss,speed_ms,0,blend_radius_m)
    movel([0.108361, -1.387591, -2.569571, -0.755227, 1.570796, 1.679158],accel_mss,speed_ms,0,blend_radius_m)
    movel([0.108712, -1.387629, -2.569543, -0.755216, 1.570796, 1.679508],accel_mss,speed_ms,0,blend_radius_m)
    movel([0.108880, -1.387836, -2.569396, -0.755158, 1.570796, 1.679677],accel_mss,speed_ms,0,blend_radius_m)
    movel([0.108710, -1.388079, -2.569222, -0.755088, 1.570796, 1.679507],accel_mss,speed_ms,0,blend_radius_m)
    movel([0.108314, -1.388273, -2.569083, -0.755033, 1.570796, 1.679110],accel_mss,speed_ms,0,blend_radius_m)
    movel([0.107973, -1.388404, -2.568989, -0.754996, 1.570796, 1.678770],accel_mss,speed_ms,0,blend_radius_m)
    speed_ms = 0.003
    movel([0.107973, -1.375417, -2.563025, -0.773946, 1.570796, 1.678770],accel_mss,speed_ms,0,blend_radius_m)
    speed_ms = 1.000
    movel([0.107973, -1.350503, -2.550705, -0.811181, 1.570796, 1.678770],accel_mss,speed_ms,0,blend_radius_m)
    movel([0.108036, -1.349102, -2.551652, -0.811635, 1.570796, 1.678832],accel_mss,speed_ms,0,blend_radius_m)
    movel([0.108036, -1.374041, -2.563990, -0.774357, 1.570796, 1.678832],accel_mss,speed_ms,0,blend_radius_m)
    speed_ms = 0.003
    movel([0.108036, -1.383759, -2.568482, -0.760148, 1.570796, 1.678832],accel_mss,speed_ms,0,blend_radius_m)
    speed_ms = 0.007
    movel([0.107706, -1.383861, -2.568410, -0.760119, 1.570796, 1.678502],accel_mss,speed_ms,0,blend_radius_m)
    movel([0.107286, -1.384012, -2.568302, -0.760075, 1.570796, 1.678082],accel_mss,speed_ms,0,blend_radius_m)
    movel([0.106844, -1.384185, -2.568179, -0.760025, 1.570796, 1.677640],accel_mss,speed_ms,0,blend_radius_m)
    movel([0.106453, -1.384354, -2.568059, -0.759976, 1.570796, 1.677249],accel_mss,speed_ms,0,blend_radius_m)
    movel([0.105610, -1.384723, -2.567796, -0.759870, 1.570796, 1.676406],accel_mss,speed_ms,0,blend_radius_m)
    movel([0.105148, -1.384885, -2.567681, -0.759823, 1.570796, 1.675944],accel_mss,speed_ms,0,blend_radius_m)
    movel([0.104900, -1.384909, -2.567664, -0.759816, 1.570796, 1.675696],accel_mss,speed_ms,0,blend_radius_m)
    movel([0.104960, -1.384453, -2.567989, -0.759948, 1.570796, 1.675757],accel_mss,speed_ms,0,blend_radius_m)
    movel([0.105494, -1.384038, -2.568284, -0.760067, 1.570796, 1.676290],accel_mss,speed_ms,0,blend_radius_m)
    movel([0.106400, -1.383572, -2.568615, -0.760202, 1.570796, 1.677196],accel_mss,speed_ms,0,blend_radius_m)
    movel([0.107695, -1.383060, -2.568978, -0.760351, 1.570796, 1.678491],accel_mss,speed_ms,0,blend_radius_m)
    movel([0.108125, -1.382914, -2.569082, -0.760393, 1.570796, 1.678921],accel_mss,speed_ms,0,blend_radius_m)
    movel([0.108375, -1.382859, -2.569121, -0.760409, 1.570796, 1.679171],accel_mss,speed_ms,0,blend_radius_m)
    movel([0.108765, -1.382928, -2.569072, -0.760389, 1.570796, 1.679562],accel_mss,speed_ms,0,blend_radius_m)
    movel([0.108980, -1.383039, -2.568993, -0.760357, 1.570796, 1.679776],accel_mss,speed_ms,0,blend_radius_m)
    movel([0.109022, -1.383237, -2.568853, -0.760299, 1.570796, 1.679819],accel_mss,speed_ms,0,blend_radius_m)
    movel([0.108786, -1.383474, -2.568684, -0.760231, 1.570796, 1.679582],accel_mss,speed_ms,0,blend_radius_m)
    movel([0.108311, -1.383674, -2.568543, -0.760173, 1.570796, 1.679107],accel_mss,speed_ms,0,blend_radius_m)
    movel([0.108036, -1.383759, -2.568482, -0.760148, 1.570796, 1.678832],accel_mss,speed_ms,0,blend_radius_m)
    speed_ms = 0.003
    movel([0.108036, -1.387042, -2.569963, -0.755384, 1.570796, 1.678832],accel_mss,speed_ms,0,blend_radius_m)
    speed_ms = 0.007
    movel([0.107706, -1.387144, -2.569890, -0.755355, 1.570796, 1.678502],accel_mss,speed_ms,0,blend_radius_m)
    movel([0.107286, -1.387296, -2.569782, -0.755312, 1.570796, 1.678082],accel_mss,speed_ms,0,blend_radius_m)
    movel([0.106844, -1.387467, -2.569659, -0.755263, 1.570796, 1.677640],accel_mss,speed_ms,0,blend_radius_m)
    movel([0.106453, -1.387636, -2.569539, -0.755215, 1.570796, 1.677249],accel_mss,speed_ms,0,blend_radius_m)
    movel([0.105610, -1.388004, -2.569275, -0.755110, 1.570796, 1.676406],accel_mss,speed_ms,0,blend_radius_m)
    movel([0.105148, -1.388165, -2.569160, -0.755064, 1.570796, 1.675944],accel_mss,speed_ms,0,blend_radius_m)
    movel([0.104900, -1.388189, -2.569143, -0.755057, 1.570796, 1.675696],accel_mss,speed_ms,0,blend_radius_m)
    movel([0.104960, -1.387735, -2.569468, -0.755186, 1.570796, 1.675757],accel_mss,speed_ms,0,blend_radius_m)
    movel([0.105494, -1.387321, -2.569764, -0.755304, 1.570796, 1.676290],accel_mss,speed_ms,0,blend_radius_m)
    movel([0.106400, -1.386856, -2.570096, -0.755437, 1.570796, 1.677196],accel_mss,speed_ms,0,blend_radius_m)
    movel([0.107695, -1.386346, -2.570460, -0.755583, 1.570796, 1.678491],accel_mss,speed_ms,0,blend_radius_m)
    movel([0.108125, -1.386200, -2.570564, -0.755625, 1.570796, 1.678921],accel_mss,speed_ms,0,blend_radius_m)
    movel([0.108375, -1.386145, -2.570603, -0.755641, 1.570796, 1.679171],accel_mss,speed_ms,0,blend_radius_m)
    movel([0.108765, -1.386214, -2.570554, -0.755621, 1.570796, 1.679562],accel_mss,speed_ms,0,blend_radius_m)
    movel([0.108980, -1.386325, -2.570475, -0.755589, 1.570796, 1.679776],accel_mss,speed_ms,0,blend_radius_m)
    movel([0.109022, -1.386522, -2.570334, -0.755533, 1.570796, 1.679819],accel_mss,speed_ms,0,blend_radius_m)
    movel([0.108786, -1.386759, -2.570165, -0.755465, 1.570796, 1.679582],accel_mss,speed_ms,0,blend_radius_m)
    movel([0.108311, -1.386958, -2.570023, -0.755408, 1.570796, 1.679107],accel_mss,speed_ms,0,blend_radius_m)
    movel([0.108036, -1.387042, -2.569963, -0.755384, 1.570796, 1.678832],accel_mss,speed_ms,0,blend_radius_m)
    speed_ms = 0.003
    movel([0.108036, -1.374041, -2.563990, -0.774357, 1.570796, 1.678832],accel_mss,speed_ms,0,blend_radius_m)
    speed_ms = 1.000
    movel([0.108036, -1.349102, -2.551652, -0.811635, 1.570796, 1.678832],accel_mss,speed_ms,0,blend_radius_m)
    movel([0.108046, -1.347695, -2.552600, -0.812094, 1.570796, 1.678842],accel_mss,speed_ms,0,blend_radius_m)
    movel([0.108046, -1.372660, -2.564956, -0.774773, 1.570796, 1.678842],accel_mss,speed_ms,0,blend_radius_m)
    speed_ms = 0.003
    movel([0.108046, -1.382388, -2.569455, -0.760546, 1.570796, 1.678842],accel_mss,speed_ms,0,blend_radius_m)
    speed_ms = 0.007
    movel([0.107493, -1.382574, -2.569323, -0.760492, 1.570796, 1.678290],accel_mss,speed_ms,0,blend_radius_m)
    movel([0.106983, -1.382746, -2.569201, -0.760442, 1.570796, 1.677780],accel_mss,speed_ms,0,blend_radius_m)
    movel([0.106468, -1.382941, -2.569063, -0.760385, 1.570796, 1.677264],accel_mss,speed_ms,0,blend_radius_m)
    movel([0.106014, -1.383128, -2.568930, -0.760331, 1.570796, 1.676811],accel_mss,speed_ms,0,blend_radius_m)
    movel([0.105727, -1.383271, -2.568828, -0.760289, 1.570796, 1.676524],accel_mss,speed_ms,0,blend_radius_m)
    movel([0.105343, -1.383462, -2.568693, -0.760234, 1.570796, 1.676139],accel_mss,speed_ms,0,blend_radius_m)
    movel([0.104988, -1.383409, -2.568731, -0.760249, 1.570796, 1.675785],accel_mss,speed_ms,0,blend_radius_m)
    movel([0.104973, -1.383177, -2.568895, -0.760317, 1.570796, 1.675770],accel_mss,speed_ms,0,blend_radius_m)
    movel([0.105166, -1.382821, -2.569148, -0.760420, 1.570796, 1.675962],accel_mss,speed_ms,0,blend_radius_m)
    movel([0.105621, -1.382469, -2.569397, -0.760522, 1.570796, 1.676417],accel_mss,speed_ms,0,blend_radius_m)
    movel([0.106415, -1.382080, -2.569673, -0.760636, 1.570796, 1.677212],accel_mss,speed_ms,0,blend_radius_m)
    movel([0.107697, -1.381596, -2.570015, -0.760777, 1.570796, 1.678493],accel_mss,speed_ms,0,blend_radius_m)
    movel([0.108165, -1.381440, -2.570126, -0.760823, 1.570796, 1.678961],accel_mss,speed_ms,0,blend_radius_m)
    movel([0.108430, -1.381380, -2.570169, -0.760841, 1.570796, 1.679226],accel_mss,speed_ms,0,blend_radius_m)
    movel([0.108831, -1.381447, -2.570121, -0.760821, 1.570796, 1.679627],accel_mss,speed_ms,0,blend_radius_m)
    movel([0.109048, -1.381564, -2.570039, -0.760787, 1.570796, 1.679844],accel_mss,speed_ms,0,blend_radius_m)
    movel([0.109077, -1.381790, -2.569878, -0.760721, 1.570796, 1.679873],accel_mss,speed_ms,0,blend_radius_m)
    movel([0.108772, -1.382086, -2.569669, -0.760634, 1.570796, 1.679569],accel_mss,speed_ms,0,blend_radius_m)
    movel([0.108466, -1.382226, -2.569570, -0.760593, 1.570796, 1.679262],accel_mss,speed_ms,0,blend_radius_m)
    movel([0.108046, -1.382388, -2.569455, -0.760546, 1.570796, 1.678842],accel_mss,speed_ms,0,blend_radius_m)
    speed_ms = 0.003
    movel([0.108046, -1.385676, -2.570938, -0.755776, 1.570796, 1.678842],accel_mss,speed_ms,0,blend_radius_m)
    speed_ms = 0.007
    movel([0.107493, -1.385861, -2.570805, -0.755722, 1.570796, 1.678290],accel_mss,speed_ms,0,blend_radius_m)
    movel([0.106983, -1.386033, -2.570683, -0.755673, 1.570796, 1.677780],accel_mss,speed_ms,0,blend_radius_m)
    movel([0.106468, -1.386227, -2.570544, -0.755617, 1.570796, 1.677264],accel_mss,speed_ms,0,blend_radius_m)
    movel([0.106014, -1.386413, -2.570412, -0.755564, 1.570796, 1.676811],accel_mss,speed_ms,0,blend_radius_m)
    movel([0.105727, -1.386556, -2.570310, -0.755523, 1.570796, 1.676524],accel_mss,speed_ms,0,blend_radius_m)
    movel([0.105343, -1.386746, -2.570174, -0.755469, 1.570796, 1.676139],accel_mss,speed_ms,0,blend_radius_m)
    movel([0.104988, -1.386693, -2.570212, -0.755484, 1.570796, 1.675785],accel_mss,speed_ms,0,blend_radius_m)
    movel([0.104973, -1.386462, -2.570377, -0.755550, 1.570796, 1.675770],accel_mss,speed_ms,0,blend_radius_m)
    movel([0.105166, -1.386108, -2.570630, -0.755652, 1.570796, 1.675962],accel_mss,speed_ms,0,blend_radius_m)
    movel([0.105621, -1.385756, -2.570880, -0.755753, 1.570796, 1.676417],accel_mss,speed_ms,0,blend_radius_m)
    movel([0.106415, -1.385369, -2.571156, -0.755864, 1.570796, 1.677212],accel_mss,speed_ms,0,blend_radius_m)
    movel([0.107697, -1.384886, -2.571499, -0.756003, 1.570796, 1.678493],accel_mss,speed_ms,0,blend_radius_m)
    movel([0.108165, -1.384730, -2.571611, -0.756049, 1.570796, 1.678961],accel_mss,speed_ms,0,blend_radius_m)
    movel([0.108430, -1.384670, -2.571653, -0.756066, 1.570796, 1.679226],accel_mss,speed_ms,0,blend_radius_m)
    movel([0.108831, -1.384737, -2.571606, -0.756047, 1.570796, 1.679627],accel_mss,speed_ms,0,blend_radius_m)
    movel([0.109048, -1.384853, -2.571523, -0.756013, 1.570796, 1.679844],accel_mss,speed_ms,0,blend_radius_m)
    movel([0.109077, -1.385079, -2.571362, -0.755948, 1.570796, 1.679873],accel_mss,speed_ms,0,blend_radius_m)
    movel([0.108772, -1.385374, -2.571152, -0.755863, 1.570796, 1.679569],accel_mss,speed_ms,0,blend_radius_m)
    movel([0.108466, -1.385514, -2.571053, -0.755822, 1.570796, 1.679262],accel_mss,speed_ms,0,blend_radius_m)
    movel([0.108046, -1.385676, -2.570938, -0.755776, 1.570796, 1.678842],accel_mss,speed_ms,0,blend_radius_m)
    speed_ms = 0.003
    movel([0.108046, -1.372660, -2.564956, -0.774773, 1.570796, 1.678842],accel_mss,speed_ms,0,blend_radius_m)
    speed_ms = 1.000
    movel([0.108046, -1.347695, -2.552600, -0.812094, 1.570796, 1.678842],accel_mss,speed_ms,0,blend_radius_m)
    movel([0.107957, -1.346153, -2.553637, -0.812600, 1.570796, 1.678753],accel_mss,speed_ms,0,blend_radius_m)
    movel([0.107957, -1.371145, -2.566013, -0.775232, 1.570796, 1.678753],accel_mss,speed_ms,0,blend_radius_m)
    speed_ms = 0.003
    movel([0.107957, -1.380885, -2.570519, -0.760986, 1.570796, 1.678753],accel_mss,speed_ms,0,blend_radius_m)
    speed_ms = 0.007
    movel([0.107460, -1.381077, -2.570383, -0.760929, 1.570796, 1.678256],accel_mss,speed_ms,0,blend_radius_m)
    movel([0.106951, -1.381270, -2.570246, -0.760873, 1.570796, 1.677748],accel_mss,speed_ms,0,blend_radius_m)
    movel([0.106468, -1.381455, -2.570116, -0.760819, 1.570796, 1.677264],accel_mss,speed_ms,0,blend_radius_m)
    movel([0.106060, -1.381617, -2.570001, -0.760771, 1.570796, 1.676856],accel_mss,speed_ms,0,blend_radius_m)
    movel([0.105690, -1.381764, -2.569897, -0.760728, 1.570796, 1.676486],accel_mss,speed_ms,0,blend_radius_m)
    movel([0.105469, -1.381660, -2.569971, -0.760759, 1.570796, 1.676265],accel_mss,speed_ms,0,blend_radius_m)
    movel([0.105525, -1.381301, -2.570224, -0.760864, 1.570796, 1.676321],accel_mss,speed_ms,0,blend_radius_m)
    movel([0.105823, -1.380972, -2.570457, -0.760960, 1.570796, 1.676619],accel_mss,speed_ms,0,blend_radius_m)
    movel([0.106443, -1.380643, -2.570689, -0.761057, 1.570796, 1.677239],accel_mss,speed_ms,0,blend_radius_m)
    movel([0.107505, -1.380266, -2.570955, -0.761167, 1.570796, 1.678302],accel_mss,speed_ms,0,blend_radius_m)
    movel([0.108170, -1.380061, -2.571100, -0.761228, 1.570796, 1.678967],accel_mss,speed_ms,0,blend_radius_m)
    movel([0.108524, -1.379975, -2.571160, -0.761253, 1.570796, 1.679320],accel_mss,speed_ms,0,blend_radius_m)
    movel([0.108896, -1.380010, -2.571136, -0.761243, 1.570796, 1.679692],accel_mss,speed_ms,0,blend_radius_m)
    movel([0.109065, -1.380218, -2.570989, -0.761182, 1.570796, 1.679862],accel_mss,speed_ms,0,blend_radius_m)
    movel([0.108895, -1.380457, -2.570821, -0.761111, 1.570796, 1.679692],accel_mss,speed_ms,0,blend_radius_m)
    movel([0.108402, -1.380701, -2.570649, -0.761040, 1.570796, 1.679198],accel_mss,speed_ms,0,blend_radius_m)
    movel([0.107957, -1.380885, -2.570519, -0.760986, 1.570796, 1.678753],accel_mss,speed_ms,0,blend_radius_m)
    speed_ms = 0.003
    movel([0.107957, -1.384176, -2.572004, -0.756209, 1.570796, 1.678753],accel_mss,speed_ms,0,blend_radius_m)
    speed_ms = 0.007
    movel([0.107460, -1.384368, -2.571868, -0.756153, 1.570796, 1.678256],accel_mss,speed_ms,0,blend_radius_m)
    movel([0.106951, -1.384561, -2.571731, -0.756097, 1.570796, 1.677748],accel_mss,speed_ms,0,blend_radius_m)
    movel([0.106468, -1.384745, -2.571600, -0.756044, 1.570796, 1.677264],accel_mss,speed_ms,0,blend_radius_m)
    movel([0.106060, -1.384907, -2.571485, -0.755998, 1.570796, 1.676856],accel_mss,speed_ms,0,blend_radius_m)
    movel([0.105690, -1.385054, -2.571380, -0.755955, 1.570796, 1.676486],accel_mss,speed_ms,0,blend_radius_m)
    movel([0.105469, -1.384949, -2.571454, -0.755985, 1.570796, 1.676265],accel_mss,speed_ms,0,blend_radius_m)
    movel([0.105525, -1.384592, -2.571709, -0.756089, 1.570796, 1.676321],accel_mss,speed_ms,0,blend_radius_m)
    movel([0.105823, -1.384264, -2.571942, -0.756184, 1.570796, 1.676619],accel_mss,speed_ms,0,blend_radius_m)
    movel([0.106443, -1.383935, -2.572175, -0.756279, 1.570796, 1.677239],accel_mss,speed_ms,0,blend_radius_m)
    movel([0.107505, -1.383559, -2.572442, -0.756388, 1.570796, 1.678302],accel_mss,speed_ms,0,blend_radius_m)
    movel([0.108170, -1.383355, -2.572586, -0.756447, 1.570796, 1.678967],accel_mss,speed_ms,0,blend_radius_m)
    movel([0.108524, -1.383269, -2.572647, -0.756472, 1.570796, 1.679320],accel_mss,speed_ms,0,blend_radius_m)
    movel([0.108896, -1.383304, -2.572622, -0.756462, 1.570796, 1.679692],accel_mss,speed_ms,0,blend_radius_m)
    movel([0.109065, -1.383511, -2.572476, -0.756402, 1.570796, 1.679862],accel_mss,speed_ms,0,blend_radius_m)
    movel([0.108895, -1.383750, -2.572306, -0.756333, 1.570796, 1.679692],accel_mss,speed_ms,0,blend_radius_m)
    movel([0.108402, -1.383993, -2.572134, -0.756262, 1.570796, 1.679198],accel_mss,speed_ms,0,blend_radius_m)
    movel([0.107957, -1.384176, -2.572004, -0.756209, 1.570796, 1.678753],accel_mss,speed_ms,0,blend_radius_m)
    speed_ms = 0.003
    movel([0.107957, -1.371145, -2.566013, -0.775232, 1.570796, 1.678753],accel_mss,speed_ms,0,blend_radius_m)
    speed_ms = 1.000
    movel([0.107957, -1.346153, -2.553637, -0.812600, 1.570796, 1.678753],accel_mss,speed_ms,0,blend_radius_m)
    movel([0.107938, -1.344656, -2.554639, -0.813093, 1.570796, 1.678735],accel_mss,speed_ms,0,blend_radius_m)
    movel([0.107938, -1.369675, -2.567035, -0.775680, 1.570796, 1.678735],accel_mss,speed_ms,0,blend_radius_m)
    speed_ms = 0.003
    movel([0.107938, -1.379426, -2.571548, -0.761415, 1.570796, 1.678735],accel_mss,speed_ms,0,blend_radius_m)
    speed_ms = 0.007
    movel([0.107342, -1.379621, -2.571410, -0.761358, 1.570796, 1.678138],accel_mss,speed_ms,0,blend_radius_m)
    movel([0.107347, -1.379363, -2.571592, -0.761434, 1.570796, 1.678143],accel_mss,speed_ms,0,blend_radius_m)
    movel([0.107964, -1.378932, -2.571896, -0.761562, 1.570796, 1.678760],accel_mss,speed_ms,0,blend_radius_m)
    movel([0.108387, -1.378656, -2.572089, -0.761643, 1.570796, 1.679184],accel_mss,speed_ms,0,blend_radius_m)
    movel([0.108732, -1.378526, -2.572181, -0.761682, 1.570796, 1.679529],accel_mss,speed_ms,0,blend_radius_m)
    movel([0.108975, -1.378670, -2.572080, -0.761639, 1.570796, 1.679772],accel_mss,speed_ms,0,blend_radius_m)
    movel([0.108836, -1.379009, -2.571842, -0.761539, 1.570796, 1.679632],accel_mss,speed_ms,0,blend_radius_m)
    movel([0.108501, -1.379192, -2.571712, -0.761484, 1.570796, 1.679298],accel_mss,speed_ms,0,blend_radius_m)
    movel([0.108228, -1.379313, -2.571627, -0.761449, 1.570796, 1.679024],accel_mss,speed_ms,0,blend_radius_m)
    movel([0.107938, -1.379426, -2.571548, -0.761415, 1.570796, 1.678735],accel_mss,speed_ms,0,blend_radius_m)
    speed_ms = 0.003
    movel([0.107938, -1.382722, -2.573035, -0.756632, 1.570796, 1.678735],accel_mss,speed_ms,0,blend_radius_m)
    speed_ms = 0.007
    movel([0.107342, -1.382916, -2.572898, -0.756575, 1.570796, 1.678138],accel_mss,speed_ms,0,blend_radius_m)
    movel([0.107347, -1.382659, -2.573079, -0.756650, 1.570796, 1.678143],accel_mss,speed_ms,0,blend_radius_m)
    movel([0.107964, -1.382229, -2.573384, -0.756776, 1.570796, 1.678760],accel_mss,speed_ms,0,blend_radius_m)
    movel([0.108387, -1.381954, -2.573578, -0.756857, 1.570796, 1.679184],accel_mss,speed_ms,0,blend_radius_m)
    movel([0.108732, -1.381824, -2.573670, -0.756895, 1.570796, 1.679529],accel_mss,speed_ms,0,blend_radius_m)
    movel([0.108975, -1.381968, -2.573569, -0.756853, 1.570796, 1.679772],accel_mss,speed_ms,0,blend_radius_m)
    movel([0.108836, -1.382305, -2.573330, -0.756754, 1.570796, 1.679632],accel_mss,speed_ms,0,blend_radius_m)
    movel([0.108501, -1.382489, -2.573200, -0.756700, 1.570796, 1.679298],accel_mss,speed_ms,0,blend_radius_m)
    movel([0.108228, -1.382609, -2.573115, -0.756665, 1.570796, 1.679024],accel_mss,speed_ms,0,blend_radius_m)
    movel([0.107938, -1.382722, -2.573035, -0.756632, 1.570796, 1.678735],accel_mss,speed_ms,0,blend_radius_m)
    speed_ms = 0.003
    movel([0.107938, -1.369675, -2.567035, -0.775680, 1.570796, 1.678735],accel_mss,speed_ms,0,blend_radius_m)
    speed_ms = 1.000
    movel([0.107938, -1.344656, -2.554639, -0.813093, 1.570796, 1.678735],accel_mss,speed_ms,0,blend_radius_m)
    movel([0.107459, -1.343867, -2.555167, -0.813355, 1.570796, 1.678255],accel_mss,speed_ms,0,blend_radius_m)
    movel([0.107459, -1.368899, -2.567572, -0.775917, 1.570796, 1.678255],accel_mss,speed_ms,0,blend_radius_m)
    speed_ms = 0.003
    movel([0.107459, -1.378656, -2.572089, -0.761643, 1.570796, 1.678255],accel_mss,speed_ms,0,blend_radius_m)
    speed_ms = 0.007
    movel([0.106787, -1.379080, -2.571791, -0.761518, 1.570796, 1.677584],accel_mss,speed_ms,0,blend_radius_m)
    movel([0.106338, -1.379277, -2.571652, -0.761459, 1.570796, 1.677134],accel_mss,speed_ms,0,blend_radius_m)
    movel([0.106106, -1.379255, -2.571668, -0.761466, 1.570796, 1.676902],accel_mss,speed_ms,0,blend_radius_m)
    movel([0.106047, -1.379065, -2.571802, -0.761522, 1.570796, 1.676843],accel_mss,speed_ms,0,blend_radius_m)
    movel([0.106228, -1.377942, -2.572592, -0.761856, 1.570796, 1.677025],accel_mss,speed_ms,0,blend_radius_m)
    movel([0.106395, -1.376860, -2.573350, -0.762179, 1.570796, 1.677191],accel_mss,speed_ms,0,blend_radius_m)
    movel([0.106578, -1.375631, -2.574211, -0.762547, 1.570796, 1.677374],accel_mss,speed_ms,0,blend_radius_m)
    movel([0.106821, -1.374030, -2.575328, -0.763031, 1.570796, 1.677617],accel_mss,speed_ms,0,blend_radius_m)
    movel([0.106988, -1.373093, -2.575980, -0.763316, 1.570796, 1.677784],accel_mss,speed_ms,0,blend_radius_m)
    movel([0.107121, -1.372467, -2.576415, -0.763507, 1.570796, 1.677917],accel_mss,speed_ms,0,blend_radius_m)
    movel([0.107666, -1.372082, -2.576682, -0.763625, 1.570796, 1.678462],accel_mss,speed_ms,0,blend_radius_m)
    movel([0.108309, -1.372101, -2.576669, -0.763619, 1.570796, 1.679105],accel_mss,speed_ms,0,blend_radius_m)
    movel([0.108956, -1.372304, -2.576528, -0.763557, 1.570796, 1.679752],accel_mss,speed_ms,0,blend_radius_m)
    movel([0.109432, -1.372658, -2.576282, -0.763449, 1.570796, 1.680228],accel_mss,speed_ms,0,blend_radius_m)
    movel([0.109711, -1.373202, -2.575904, -0.763283, 1.570796, 1.680507],accel_mss,speed_ms,0,blend_radius_m)
    movel([0.109808, -1.374012, -2.575341, -0.763037, 1.570796, 1.680604],accel_mss,speed_ms,0,blend_radius_m)
    movel([0.109726, -1.375002, -2.574650, -0.762737, 1.570796, 1.680523],accel_mss,speed_ms,0,blend_radius_m)
    movel([0.109459, -1.376100, -2.573883, -0.762407, 1.570796, 1.680255],accel_mss,speed_ms,0,blend_radius_m)
    movel([0.109156, -1.376853, -2.573355, -0.762181, 1.570796, 1.679952],accel_mss,speed_ms,0,blend_radius_m)
    movel([0.108739, -1.377506, -2.572897, -0.761985, 1.570796, 1.679536],accel_mss,speed_ms,0,blend_radius_m)
    movel([0.108184, -1.378094, -2.572485, -0.761810, 1.570796, 1.678981],accel_mss,speed_ms,0,blend_radius_m)
    movel([0.107459, -1.378656, -2.572089, -0.761643, 1.570796, 1.678255],accel_mss,speed_ms,0,blend_radius_m)
    speed_ms = 0.003
    movel([0.107459, -1.381954, -2.573578, -0.756857, 1.570796, 1.678255],accel_mss,speed_ms,0,blend_radius_m)
    speed_ms = 0.007
    movel([0.106787, -1.382377, -2.573279, -0.756733, 1.570796, 1.677584],accel_mss,speed_ms,0,blend_radius_m)
    movel([0.106338, -1.382573, -2.573140, -0.756676, 1.570796, 1.677134],accel_mss,speed_ms,0,blend_radius_m)
    movel([0.106106, -1.382551, -2.573156, -0.756682, 1.570796, 1.676902],accel_mss,speed_ms,0,blend_radius_m)
    movel([0.106047, -1.382362, -2.573290, -0.756737, 1.570796, 1.676843],accel_mss,speed_ms,0,blend_radius_m)
    movel([0.106228, -1.381241, -2.574082, -0.757066, 1.570796, 1.677025],accel_mss,speed_ms,0,blend_radius_m)
    movel([0.106395, -1.380163, -2.574842, -0.757384, 1.570796, 1.677191],accel_mss,speed_ms,0,blend_radius_m)
    movel([0.106578, -1.378937, -2.575704, -0.757748, 1.570796, 1.677374],accel_mss,speed_ms,0,blend_radius_m)
    movel([0.106821, -1.377340, -2.576824, -0.758225, 1.570796, 1.677617],accel_mss,speed_ms,0,blend_radius_m)
    movel([0.106988, -1.376405, -2.577478, -0.758505, 1.570796, 1.677784],accel_mss,speed_ms,0,blend_radius_m)
    movel([0.107121, -1.375781, -2.577914, -0.758694, 1.570796, 1.677917],accel_mss,speed_ms,0,blend_radius_m)
    movel([0.107666, -1.375398, -2.578182, -0.758810, 1.570796, 1.678462],accel_mss,speed_ms,0,blend_radius_m)
    movel([0.108309, -1.375417, -2.578168, -0.758804, 1.570796, 1.679105],accel_mss,speed_ms,0,blend_radius_m)
    movel([0.108956, -1.375619, -2.578027, -0.758743, 1.570796, 1.679752],accel_mss,speed_ms,0,blend_radius_m)
    movel([0.109432, -1.375972, -2.577781, -0.758636, 1.570796, 1.680228],accel_mss,speed_ms,0,blend_radius_m)
    movel([0.109711, -1.376515, -2.577402, -0.758473, 1.570796, 1.680507],accel_mss,speed_ms,0,blend_radius_m)
    movel([0.109808, -1.377322, -2.576837, -0.758230, 1.570796, 1.680604],accel_mss,speed_ms,0,blend_radius_m)
    movel([0.109726, -1.378310, -2.576144, -0.757935, 1.570796, 1.680523],accel_mss,speed_ms,0,blend_radius_m)
    movel([0.109459, -1.379404, -2.575376, -0.757609, 1.570796, 1.680255],accel_mss,speed_ms,0,blend_radius_m)
    movel([0.109156, -1.380156, -2.574847, -0.757386, 1.570796, 1.679952],accel_mss,speed_ms,0,blend_radius_m)
    movel([0.108739, -1.380807, -2.574388, -0.757194, 1.570796, 1.679536],accel_mss,speed_ms,0,blend_radius_m)
    movel([0.108184, -1.381393, -2.573975, -0.757021, 1.570796, 1.678981],accel_mss,speed_ms,0,blend_radius_m)
    movel([0.107459, -1.381954, -2.573578, -0.756857, 1.570796, 1.678255],accel_mss,speed_ms,0,blend_radius_m)
    speed_ms = 0.003
    movel([0.107459, -1.368899, -2.567572, -0.775917, 1.570796, 1.678255],accel_mss,speed_ms,0,blend_radius_m)
    speed_ms = 1.000
    movel([0.107459, -1.343867, -2.555167, -0.813355, 1.570796, 1.678255],accel_mss,speed_ms,0,blend_radius_m)
    movel([0.112766, -1.336699, -2.559921, -0.815769, 1.570796, 1.683562],accel_mss,speed_ms,0,blend_radius_m)
    movel([0.112766, -1.361858, -2.572418, -0.778114, 1.570796, 1.683562],accel_mss,speed_ms,0,blend_radius_m)
    speed_ms = 0.003
    movel([0.112766, -1.371669, -2.576969, -0.763751, 1.570796, 1.683562],accel_mss,speed_ms,0,blend_radius_m)
    speed_ms = 0.007
    movel([0.112640, -1.371423, -2.577139, -0.763827, 1.570796, 1.683436],accel_mss,speed_ms,0,blend_radius_m)
    movel([0.112664, -1.370800, -2.577571, -0.764018, 1.570796, 1.683461],accel_mss,speed_ms,0,blend_radius_m)
    movel([0.112748, -1.369984, -2.578135, -0.764270, 1.570796, 1.683545],accel_mss,speed_ms,0,blend_radius_m)
    movel([0.114064, -1.369651, -2.578365, -0.764373, 1.570796, 1.684861],accel_mss,speed_ms,0,blend_radius_m)
    movel([0.115040, -1.369430, -2.578518, -0.764442, 1.570796, 1.685836],accel_mss,speed_ms,0,blend_radius_m)
    movel([0.115513, -1.369409, -2.578532, -0.764448, 1.570796, 1.686309],accel_mss,speed_ms,0,blend_radius_m)
    movel([0.115676, -1.369559, -2.578429, -0.764401, 1.570796, 1.686472],accel_mss,speed_ms,0,blend_radius_m)
    movel([0.115615, -1.369869, -2.578214, -0.764305, 1.570796, 1.686411],accel_mss,speed_ms,0,blend_radius_m)
    movel([0.115514, -1.370131, -2.578033, -0.764225, 1.570796, 1.686311],accel_mss,speed_ms,0,blend_radius_m)
    movel([0.115438, -1.370635, -2.577685, -0.764069, 1.570796, 1.686234],accel_mss,speed_ms,0,blend_radius_m)
    movel([0.115115, -1.370976, -2.577449, -0.763964, 1.570796, 1.685911],accel_mss,speed_ms,0,blend_radius_m)
    movel([0.114542, -1.371299, -2.577225, -0.763865, 1.570796, 1.685338],accel_mss,speed_ms,0,blend_radius_m)
    movel([0.113790, -1.371559, -2.577045, -0.763785, 1.570796, 1.684586],accel_mss,speed_ms,0,blend_radius_m)
    movel([0.113081, -1.371719, -2.576934, -0.763736, 1.570796, 1.683877],accel_mss,speed_ms,0,blend_radius_m)
    movel([0.112766, -1.371669, -2.576969, -0.763751, 1.570796, 1.683562],accel_mss,speed_ms,0,blend_radius_m)
    speed_ms = 0.003
    movel([0.112766, -1.374985, -2.578469, -0.758934, 1.570796, 1.683562],accel_mss,speed_ms,0,blend_radius_m)
    speed_ms = 0.007
    movel([0.112640, -1.374740, -2.578640, -0.759009, 1.570796, 1.683436],accel_mss,speed_ms,0,blend_radius_m)
    movel([0.112664, -1.374119, -2.579072, -0.759198, 1.570796, 1.683461],accel_mss,speed_ms,0,blend_radius_m)
    movel([0.112748, -1.373305, -2.579638, -0.759446, 1.570796, 1.683545],accel_mss,speed_ms,0,blend_radius_m)
    movel([0.114064, -1.372973, -2.579869, -0.759547, 1.570796, 1.684861],accel_mss,speed_ms,0,blend_radius_m)
    movel([0.115040, -1.372752, -2.580022, -0.759615, 1.570796, 1.685836],accel_mss,speed_ms,0,blend_radius_m)
    movel([0.115513, -1.372732, -2.580036, -0.759621, 1.570796, 1.686309],accel_mss,speed_ms,0,blend_radius_m)
    movel([0.115676, -1.372881, -2.579932, -0.759576, 1.570796, 1.686472],accel_mss,speed_ms,0,blend_radius_m)
    movel([0.115615, -1.373191, -2.579717, -0.759481, 1.570796, 1.686411],accel_mss,speed_ms,0,blend_radius_m)
    movel([0.115514, -1.373452, -2.579536, -0.759401, 1.570796, 1.686311],accel_mss,speed_ms,0,blend_radius_m)
    movel([0.115438, -1.373954, -2.579187, -0.759248, 1.570796, 1.686234],accel_mss,speed_ms,0,blend_radius_m)
    movel([0.115115, -1.374294, -2.578951, -0.759144, 1.570796, 1.685911],accel_mss,speed_ms,0,blend_radius_m)
    movel([0.114542, -1.374617, -2.578726, -0.759046, 1.570796, 1.685338],accel_mss,speed_ms,0,blend_radius_m)
    movel([0.113790, -1.374876, -2.578545, -0.758968, 1.570796, 1.684586],accel_mss,speed_ms,0,blend_radius_m)
    movel([0.113081, -1.375035, -2.578434, -0.758919, 1.570796, 1.683877],accel_mss,speed_ms,0,blend_radius_m)
    movel([0.112766, -1.374985, -2.578469, -0.758934, 1.570796, 1.683562],accel_mss,speed_ms,0,blend_radius_m)
    speed_ms = 0.003
    movel([0.112766, -1.361858, -2.572418, -0.778114, 1.570796, 1.683562],accel_mss,speed_ms,0,blend_radius_m)
    speed_ms = 1.000
    movel([0.112766, -1.336699, -2.559921, -0.815769, 1.570796, 1.683562],accel_mss,speed_ms,0,blend_radius_m)
    movel([0.113433, -1.334323, -2.561482, -0.816584, 1.570796, 1.684229],accel_mss,speed_ms,0,blend_radius_m)
    movel([0.113433, -1.359522, -2.574009, -0.778858, 1.570796, 1.684229],accel_mss,speed_ms,0,blend_radius_m)
    speed_ms = 0.003
    movel([0.113433, -1.369351, -2.578572, -0.764466, 1.570796, 1.684229],accel_mss,speed_ms,0,blend_radius_m)
    speed_ms = 0.007
    movel([0.113200, -1.369116, -2.578734, -0.764539, 1.570796, 1.683996],accel_mss,speed_ms,0,blend_radius_m)
    movel([0.113209, -1.368786, -2.578962, -0.764641, 1.570796, 1.684005],accel_mss,speed_ms,0,blend_radius_m)
    movel([0.113200, -1.368460, -2.579187, -0.764743, 1.570796, 1.683996],accel_mss,speed_ms,0,blend_radius_m)
    movel([0.113074, -1.368242, -2.579336, -0.764810, 1.570796, 1.683871],accel_mss,speed_ms,0,blend_radius_m)
    movel([0.112842, -1.368148, -2.579401, -0.764840, 1.570796, 1.683639],accel_mss,speed_ms,0,blend_radius_m)
    movel([0.112523, -1.368181, -2.579379, -0.764830, 1.570796, 1.683319],accel_mss,speed_ms,0,blend_radius_m)
    movel([0.111949, -1.368213, -2.579357, -0.764820, 1.570796, 1.682746],accel_mss,speed_ms,0,blend_radius_m)
    movel([0.111243, -1.367988, -2.579512, -0.764890, 1.570796, 1.682039],accel_mss,speed_ms,0,blend_radius_m)
    movel([0.110603, -1.367616, -2.579767, -0.765006, 1.570796, 1.681399],accel_mss,speed_ms,0,blend_radius_m)
    movel([0.110212, -1.367165, -2.580077, -0.765147, 1.570796, 1.681008],accel_mss,speed_ms,0,blend_radius_m)
    movel([0.110029, -1.366891, -2.580265, -0.765233, 1.570796, 1.680825],accel_mss,speed_ms,0,blend_radius_m)
    movel([0.109878, -1.366752, -2.580361, -0.765276, 1.570796, 1.680674],accel_mss,speed_ms,0,blend_radius_m)
    movel([0.109999, -1.366376, -2.580619, -0.765394, 1.570796, 1.680795],accel_mss,speed_ms,0,blend_radius_m)
    movel([0.110066, -1.366058, -2.580837, -0.765494, 1.570796, 1.680862],accel_mss,speed_ms,0,blend_radius_m)
    movel([0.110125, -1.365664, -2.581106, -0.765618, 1.570796, 1.680922],accel_mss,speed_ms,0,blend_radius_m)
    movel([0.110214, -1.365078, -2.581508, -0.765803, 1.570796, 1.681011],accel_mss,speed_ms,0,blend_radius_m)
    movel([0.110312, -1.364717, -2.581755, -0.765918, 1.570796, 1.681108],accel_mss,speed_ms,0,blend_radius_m)
    movel([0.110471, -1.364372, -2.581990, -0.766027, 1.570796, 1.681267],accel_mss,speed_ms,0,blend_radius_m)
    movel([0.110770, -1.363875, -2.582330, -0.766185, 1.570796, 1.681566],accel_mss,speed_ms,0,blend_radius_m)
    movel([0.111001, -1.363529, -2.582566, -0.766294, 1.570796, 1.681797],accel_mss,speed_ms,0,blend_radius_m)
    movel([0.111258, -1.363172, -2.582809, -0.766408, 1.570796, 1.682054],accel_mss,speed_ms,0,blend_radius_m)
    movel([0.111508, -1.362853, -2.583026, -0.766510, 1.570796, 1.682304],accel_mss,speed_ms,0,blend_radius_m)
    movel([0.111700, -1.362635, -2.583174, -0.766579, 1.570796, 1.682497],accel_mss,speed_ms,0,blend_radius_m)
    movel([0.112170, -1.362219, -2.583458, -0.766713, 1.570796, 1.682966],accel_mss,speed_ms,0,blend_radius_m)
    movel([0.112837, -1.361736, -2.583786, -0.766867, 1.570796, 1.683634],accel_mss,speed_ms,0,blend_radius_m)
    movel([0.113532, -1.361295, -2.584086, -0.767009, 1.570796, 1.684329],accel_mss,speed_ms,0,blend_radius_m)
    movel([0.114080, -1.361022, -2.584271, -0.767097, 1.570796, 1.684876],accel_mss,speed_ms,0,blend_radius_m)
    movel([0.114439, -1.360855, -2.584384, -0.767150, 1.570796, 1.685235],accel_mss,speed_ms,0,blend_radius_m)
    movel([0.114838, -1.360572, -2.584576, -0.767242, 1.570796, 1.685635],accel_mss,speed_ms,0,blend_radius_m)
    movel([0.115414, -1.360389, -2.584700, -0.767301, 1.570796, 1.686211],accel_mss,speed_ms,0,blend_radius_m)
    movel([0.115941, -1.360262, -2.584785, -0.767341, 1.570796, 1.686737],accel_mss,speed_ms,0,blend_radius_m)
    movel([0.116093, -1.360400, -2.584692, -0.767297, 1.570796, 1.686889],accel_mss,speed_ms,0,blend_radius_m)
    movel([0.116466, -1.360370, -2.584712, -0.767307, 1.570796, 1.687262],accel_mss,speed_ms,0,blend_radius_m)
    movel([0.117091, -1.360338, -2.584734, -0.767317, 1.570796, 1.687887],accel_mss,speed_ms,0,blend_radius_m)
    movel([0.117773, -1.360429, -2.584672, -0.767288, 1.570796, 1.688569],accel_mss,speed_ms,0,blend_radius_m)
    movel([0.118423, -1.360624, -2.584540, -0.767225, 1.570796, 1.689219],accel_mss,speed_ms,0,blend_radius_m)
    movel([0.118955, -1.360908, -2.584348, -0.767133, 1.570796, 1.689751],accel_mss,speed_ms,0,blend_radius_m)
    movel([0.119345, -1.361234, -2.584126, -0.767028, 1.570796, 1.690142],accel_mss,speed_ms,0,blend_radius_m)
    movel([0.119677, -1.361646, -2.583847, -0.766896, 1.570796, 1.690474],accel_mss,speed_ms,0,blend_radius_m)
    movel([0.119903, -1.362061, -2.583565, -0.766763, 1.570796, 1.690699],accel_mss,speed_ms,0,blend_radius_m)
    movel([0.119940, -1.362378, -2.583349, -0.766661, 1.570796, 1.690737],accel_mss,speed_ms,0,blend_radius_m)
    movel([0.119963, -1.362607, -2.583194, -0.766588, 1.570796, 1.690759],accel_mss,speed_ms,0,blend_radius_m)
    movel([0.120018, -1.362814, -2.583053, -0.766522, 1.570796, 1.690814],accel_mss,speed_ms,0,blend_radius_m)
    movel([0.119974, -1.363148, -2.582825, -0.766416, 1.570796, 1.690771],accel_mss,speed_ms,0,blend_radius_m)
    movel([0.119941, -1.363465, -2.582609, -0.766315, 1.570796, 1.690737],accel_mss,speed_ms,0,blend_radius_m)
    movel([0.120103, -1.363586, -2.582526, -0.766276, 1.570796, 1.690899],accel_mss,speed_ms,0,blend_radius_m)
    movel([0.120063, -1.363825, -2.582364, -0.766200, 1.570796, 1.690859],accel_mss,speed_ms,0,blend_radius_m)
    movel([0.119744, -1.364111, -2.582168, -0.766109, 1.570796, 1.690540],accel_mss,speed_ms,0,blend_radius_m)
    movel([0.119488, -1.364550, -2.581869, -0.765970, 1.570796, 1.690284],accel_mss,speed_ms,0,blend_radius_m)
    movel([0.118959, -1.365356, -2.581317, -0.765715, 1.570796, 1.689756],accel_mss,speed_ms,0,blend_radius_m)
    movel([0.118185, -1.366126, -2.580790, -0.765473, 1.570796, 1.688981],accel_mss,speed_ms,0,blend_radius_m)
    movel([0.117294, -1.366745, -2.580366, -0.765279, 1.570796, 1.688091],accel_mss,speed_ms,0,blend_radius_m)
    movel([0.116416, -1.367114, -2.580112, -0.765163, 1.570796, 1.687213],accel_mss,speed_ms,0,blend_radius_m)
    movel([0.116092, -1.367241, -2.580025, -0.765123, 1.570796, 1.686888],accel_mss,speed_ms,0,blend_radius_m)
    movel([0.115731, -1.367579, -2.579793, -0.765017, 1.570796, 1.686528],accel_mss,speed_ms,0,blend_radius_m)
    movel([0.115661, -1.367816, -2.579630, -0.764943, 1.570796, 1.686457],accel_mss,speed_ms,0,blend_radius_m)
    movel([0.115748, -1.368044, -2.579473, -0.764872, 1.570796, 1.686544],accel_mss,speed_ms,0,blend_radius_m)
    movel([0.115829, -1.368244, -2.579335, -0.764810, 1.570796, 1.686625],accel_mss,speed_ms,0,blend_radius_m)
    movel([0.115565, -1.368425, -2.579211, -0.764754, 1.570796, 1.686362],accel_mss,speed_ms,0,blend_radius_m)
    movel([0.115373, -1.368755, -2.578983, -0.764651, 1.570796, 1.686169],accel_mss,speed_ms,0,blend_radius_m)
    movel([0.115111, -1.368926, -2.578865, -0.764598, 1.570796, 1.685907],accel_mss,speed_ms,0,blend_radius_m)
    movel([0.114895, -1.368883, -2.578895, -0.764611, 1.570796, 1.685691],accel_mss,speed_ms,0,blend_radius_m)
    movel([0.114646, -1.368902, -2.578882, -0.764605, 1.570796, 1.685442],accel_mss,speed_ms,0,blend_radius_m)
    movel([0.114354, -1.368984, -2.578826, -0.764580, 1.570796, 1.685151],accel_mss,speed_ms,0,blend_radius_m)
    movel([0.114218, -1.368703, -2.579019, -0.764667, 1.570796, 1.685014],accel_mss,speed_ms,0,blend_radius_m)
    movel([0.114179, -1.368458, -2.579188, -0.764743, 1.570796, 1.684976],accel_mss,speed_ms,0,blend_radius_m)
    movel([0.113902, -1.368506, -2.579155, -0.764728, 1.570796, 1.684698],accel_mss,speed_ms,0,blend_radius_m)
    movel([0.113822, -1.368763, -2.578978, -0.764649, 1.570796, 1.684618],accel_mss,speed_ms,0,blend_radius_m)
    movel([0.113746, -1.369031, -2.578793, -0.764565, 1.570796, 1.684542],accel_mss,speed_ms,0,blend_radius_m)
    movel([0.113433, -1.369351, -2.578572, -0.764466, 1.570796, 1.684229],accel_mss,speed_ms,0,blend_radius_m)
    speed_ms = 0.003
    movel([0.113433, -1.372674, -2.580076, -0.759639, 1.570796, 1.684229],accel_mss,speed_ms,0,blend_radius_m)
    speed_ms = 0.007
    movel([0.113200, -1.372440, -2.580238, -0.759711, 1.570796, 1.683996],accel_mss,speed_ms,0,blend_radius_m)
    movel([0.113209, -1.372110, -2.580467, -0.759812, 1.570796, 1.684005],accel_mss,speed_ms,0,blend_radius_m)
    movel([0.113200, -1.371785, -2.580692, -0.759912, 1.570796, 1.683996],accel_mss,speed_ms,0,blend_radius_m)
    movel([0.113074, -1.371568, -2.580842, -0.759979, 1.570796, 1.683871],accel_mss,speed_ms,0,blend_radius_m)
    movel([0.112842, -1.371474, -2.580907, -0.760008, 1.570796, 1.683639],accel_mss,speed_ms,0,blend_radius_m)
    movel([0.112523, -1.371507, -2.580885, -0.759998, 1.570796, 1.683319],accel_mss,speed_ms,0,blend_radius_m)
    movel([0.111949, -1.371539, -2.580863, -0.759988, 1.570796, 1.682746],accel_mss,speed_ms,0,blend_radius_m)
    movel([0.111243, -1.371314, -2.581018, -0.760057, 1.570796, 1.682039],accel_mss,speed_ms,0,blend_radius_m)
    movel([0.110603, -1.370943, -2.581274, -0.760171, 1.570796, 1.681399],accel_mss,speed_ms,0,blend_radius_m)
    movel([0.110212, -1.370493, -2.581585, -0.760311, 1.570796, 1.681008],accel_mss,speed_ms,0,blend_radius_m)
    movel([0.110029, -1.370220, -2.581773, -0.760395, 1.570796, 1.680825],accel_mss,speed_ms,0,blend_radius_m)
    movel([0.109878, -1.370081, -2.581869, -0.760438, 1.570796, 1.680674],accel_mss,speed_ms,0,blend_radius_m)
    movel([0.109999, -1.369706, -2.582128, -0.760555, 1.570796, 1.680795],accel_mss,speed_ms,0,blend_radius_m)
    movel([0.110066, -1.369389, -2.582347, -0.760653, 1.570796, 1.680862],accel_mss,speed_ms,0,blend_radius_m)
    movel([0.110125, -1.368997, -2.582617, -0.760776, 1.570796, 1.680922],accel_mss,speed_ms,0,blend_radius_m)
    movel([0.110214, -1.368412, -2.583019, -0.760958, 1.570796, 1.681011],accel_mss,speed_ms,0,blend_radius_m)
    movel([0.110312, -1.368052, -2.583266, -0.761071, 1.570796, 1.681108],accel_mss,speed_ms,0,blend_radius_m)
    movel([0.110471, -1.367708, -2.583502, -0.761178, 1.570796, 1.681267],accel_mss,speed_ms,0,blend_radius_m)
    movel([0.110770, -1.367212, -2.583843, -0.761334, 1.570796, 1.681566],accel_mss,speed_ms,0,blend_radius_m)
    movel([0.111001, -1.366867, -2.584079, -0.761443, 1.570796, 1.681797],accel_mss,speed_ms,0,blend_radius_m)
    movel([0.111258, -1.366511, -2.584323, -0.761555, 1.570796, 1.682054],accel_mss,speed_ms,0,blend_radius_m)
    movel([0.111508, -1.366193, -2.584541, -0.761655, 1.570796, 1.682304],accel_mss,speed_ms,0,blend_radius_m)
    movel([0.111700, -1.365976, -2.584689, -0.761724, 1.570796, 1.682497],accel_mss,speed_ms,0,blend_radius_m)
    movel([0.112170, -1.365560, -2.584974, -0.761855, 1.570796, 1.682966],accel_mss,speed_ms,0,blend_radius_m)
    movel([0.112837, -1.365078, -2.585303, -0.762008, 1.570796, 1.683634],accel_mss,speed_ms,0,blend_radius_m)
    movel([0.113532, -1.364639, -2.585603, -0.762147, 1.570796, 1.684329],accel_mss,speed_ms,0,blend_radius_m)
    movel([0.114080, -1.364366, -2.585789, -0.762234, 1.570796, 1.684876],accel_mss,speed_ms,0,blend_radius_m)
    movel([0.114439, -1.364200, -2.585902, -0.762287, 1.570796, 1.685235],accel_mss,speed_ms,0,blend_radius_m)
    movel([0.114838, -1.363918, -2.586094, -0.762377, 1.570796, 1.685635],accel_mss,speed_ms,0,blend_radius_m)
    movel([0.115414, -1.363735, -2.586219, -0.762435, 1.570796, 1.686211],accel_mss,speed_ms,0,blend_radius_m)
    movel([0.115941, -1.363609, -2.586304, -0.762475, 1.570796, 1.686737],accel_mss,speed_ms,0,blend_radius_m)
    movel([0.116093, -1.363746, -2.586211, -0.762432, 1.570796, 1.686889],accel_mss,speed_ms,0,blend_radius_m)
    movel([0.116466, -1.363716, -2.586231, -0.762441, 1.570796, 1.687262],accel_mss,speed_ms,0,blend_radius_m)
    movel([0.117091, -1.363685, -2.586253, -0.762451, 1.570796, 1.687887],accel_mss,speed_ms,0,blend_radius_m)
    movel([0.117773, -1.363775, -2.586191, -0.762422, 1.570796, 1.688569],accel_mss,speed_ms,0,blend_radius_m)
    movel([0.118423, -1.363970, -2.586059, -0.762360, 1.570796, 1.689219],accel_mss,speed_ms,0,blend_radius_m)
    movel([0.118955, -1.364253, -2.585866, -0.762270, 1.570796, 1.689751],accel_mss,speed_ms,0,blend_radius_m)
    movel([0.119345, -1.364579, -2.585644, -0.762167, 1.570796, 1.690142],accel_mss,speed_ms,0,blend_radius_m)
    movel([0.119677, -1.364989, -2.585364, -0.762036, 1.570796, 1.690474],accel_mss,speed_ms,0,blend_radius_m)
    movel([0.119903, -1.365403, -2.585081, -0.761905, 1.570796, 1.690699],accel_mss,speed_ms,0,blend_radius_m)
    movel([0.119940, -1.365720, -2.584865, -0.761805, 1.570796, 1.690737],accel_mss,speed_ms,0,blend_radius_m)
    movel([0.119963, -1.365947, -2.584709, -0.761733, 1.570796, 1.690759],accel_mss,speed_ms,0,blend_radius_m)
    movel([0.120018, -1.366154, -2.584568, -0.761667, 1.570796, 1.690814],accel_mss,speed_ms,0,blend_radius_m)
    movel([0.119974, -1.366487, -2.584339, -0.761562, 1.570796, 1.690771],accel_mss,speed_ms,0,blend_radius_m)
    movel([0.119941, -1.366803, -2.584123, -0.761463, 1.570796, 1.690737],accel_mss,speed_ms,0,blend_radius_m)
    movel([0.120103, -1.366924, -2.584040, -0.761425, 1.570796, 1.690899],accel_mss,speed_ms,0,blend_radius_m)
    movel([0.120063, -1.367162, -2.583877, -0.761350, 1.570796, 1.690859],accel_mss,speed_ms,0,blend_radius_m)
    movel([0.119744, -1.367448, -2.583681, -0.761260, 1.570796, 1.690540],accel_mss,speed_ms,0,blend_radius_m)
    movel([0.119488, -1.367886, -2.583381, -0.761123, 1.570796, 1.690284],accel_mss,speed_ms,0,blend_radius_m)
    movel([0.118959, -1.368690, -2.582828, -0.760871, 1.570796, 1.689756],accel_mss,speed_ms,0,blend_radius_m)
    movel([0.118185, -1.369457, -2.582300, -0.760632, 1.570796, 1.688981],accel_mss,speed_ms,0,blend_radius_m)
    movel([0.117294, -1.370074, -2.581874, -0.760441, 1.570796, 1.688091],accel_mss,speed_ms,0,blend_radius_m)
    movel([0.116416, -1.370443, -2.581620, -0.760326, 1.570796, 1.687213],accel_mss,speed_ms,0,blend_radius_m)
    movel([0.116092, -1.370570, -2.581532, -0.760287, 1.570796, 1.686888],accel_mss,speed_ms,0,blend_radius_m)
    movel([0.115731, -1.370906, -2.581300, -0.760183, 1.570796, 1.686528],accel_mss,speed_ms,0,blend_radius_m)
    movel([0.115661, -1.371143, -2.581136, -0.760110, 1.570796, 1.686457],accel_mss,speed_ms,0,blend_radius_m)
    movel([0.115748, -1.371370, -2.580979, -0.760040, 1.570796, 1.686544],accel_mss,speed_ms,0,blend_radius_m)
    movel([0.115829, -1.371570, -2.580841, -0.759978, 1.570796, 1.686625],accel_mss,speed_ms,0,blend_radius_m)
    movel([0.115565, -1.371750, -2.580716, -0.759923, 1.570796, 1.686362],accel_mss,speed_ms,0,blend_radius_m)
    movel([0.115373, -1.372079, -2.580488, -0.759822, 1.570796, 1.686169],accel_mss,speed_ms,0,blend_radius_m)
    movel([0.115111, -1.372250, -2.580370, -0.759769, 1.570796, 1.685907],accel_mss,speed_ms,0,blend_radius_m)
    movel([0.114895, -1.372207, -2.580400, -0.759782, 1.570796, 1.685691],accel_mss,speed_ms,0,blend_radius_m)
    movel([0.114646, -1.372226, -2.580387, -0.759777, 1.570796, 1.685442],accel_mss,speed_ms,0,blend_radius_m)
    movel([0.114354, -1.372307, -2.580330, -0.759751, 1.570796, 1.685151],accel_mss,speed_ms,0,blend_radius_m)
    movel([0.114218, -1.372028, -2.580524, -0.759837, 1.570796, 1.685014],accel_mss,speed_ms,0,blend_radius_m)
    movel([0.114179, -1.371783, -2.580693, -0.759913, 1.570796, 1.684976],accel_mss,speed_ms,0,blend_radius_m)
    movel([0.113902, -1.371831, -2.580660, -0.759898, 1.570796, 1.684698],accel_mss,speed_ms,0,blend_radius_m)
    movel([0.113822, -1.372087, -2.580483, -0.759819, 1.570796, 1.684618],accel_mss,speed_ms,0,blend_radius_m)
    movel([0.113746, -1.372354, -2.580298, -0.759737, 1.570796, 1.684542],accel_mss,speed_ms,0,blend_radius_m)
    movel([0.113433, -1.372674, -2.580076, -0.759639, 1.570796, 1.684229],accel_mss,speed_ms,0,blend_radius_m)
    speed_ms = 0.003
    movel([0.113433, -1.359522, -2.574009, -0.778858, 1.570796, 1.684229],accel_mss,speed_ms,0,blend_radius_m)
    speed_ms = 1.000
    movel([0.113433, -1.334323, -2.561482, -0.816584, 1.570796, 1.684229],accel_mss,speed_ms,0,blend_radius_m)
    movel([0.114853, -1.333089, -2.562290, -0.817010, 1.570796, 1.685649],accel_mss,speed_ms,0,blend_radius_m)
    movel([0.114853, -1.358310, -2.574833, -0.779247, 1.570796, 1.685649],accel_mss,speed_ms,0,blend_radius_m)
    speed_ms = 0.003
    movel([0.114853, -1.368148, -2.579401, -0.764840, 1.570796, 1.685649],accel_mss,speed_ms,0,blend_radius_m)
    speed_ms = 0.007
    movel([0.114797, -1.367902, -2.579570, -0.764916, 1.570796, 1.685593],accel_mss,speed_ms,0,blend_radius_m)
    movel([0.114829, -1.367601, -2.579777, -0.765011, 1.570796, 1.685626],accel_mss,speed_ms,0,blend_radius_m)
    movel([0.114890, -1.367234, -2.580030, -0.765125, 1.570796, 1.685686],accel_mss,speed_ms,0,blend_radius_m)
    movel([0.115073, -1.366962, -2.580217, -0.765211, 1.570796, 1.685869],accel_mss,speed_ms,0,blend_radius_m)
    movel([0.115228, -1.367178, -2.580068, -0.765143, 1.570796, 1.686024],accel_mss,speed_ms,0,blend_radius_m)
    movel([0.115200, -1.367570, -2.579799, -0.765020, 1.570796, 1.685996],accel_mss,speed_ms,0,blend_radius_m)
    movel([0.115155, -1.367837, -2.579615, -0.764937, 1.570796, 1.685951],accel_mss,speed_ms,0,blend_radius_m)
    movel([0.115032, -1.368103, -2.579432, -0.764854, 1.570796, 1.685828],accel_mss,speed_ms,0,blend_radius_m)
    speed_ms = 0.003
    movel([0.114853, -1.371474, -2.580907, -0.760008, 1.570796, 1.685649],accel_mss,speed_ms,0,blend_radius_m)
    speed_ms = 0.007
    movel([0.114797, -1.371229, -2.581077, -0.760083, 1.570796, 1.685593],accel_mss,speed_ms,0,blend_radius_m)
    movel([0.114829, -1.370928, -2.581285, -0.760176, 1.570796, 1.685626],accel_mss,speed_ms,0,blend_radius_m)
    movel([0.114890, -1.370562, -2.581537, -0.760289, 1.570796, 1.685686],accel_mss,speed_ms,0,blend_radius_m)
    movel([0.115073, -1.370291, -2.581725, -0.760373, 1.570796, 1.685869],accel_mss,speed_ms,0,blend_radius_m)
    movel([0.115228, -1.370506, -2.581576, -0.760307, 1.570796, 1.686024],accel_mss,speed_ms,0,blend_radius_m)
    movel([0.115200, -1.370898, -2.581306, -0.760186, 1.570796, 1.685996],accel_mss,speed_ms,0,blend_radius_m)
    movel([0.115155, -1.371163, -2.581122, -0.760104, 1.570796, 1.685951],accel_mss,speed_ms,0,blend_radius_m)
    movel([0.115032, -1.371429, -2.580938, -0.760022, 1.570796, 1.685828],accel_mss,speed_ms,0,blend_radius_m)
    speed_ms = 0.003
    movel([0.114853, -1.358310, -2.574833, -0.779247, 1.570796, 1.685649],accel_mss,speed_ms,0,blend_radius_m)
    speed_ms = 1.000
    movel([0.114853, -1.333089, -2.562290, -0.817010, 1.570796, 1.685649],accel_mss,speed_ms,0,blend_radius_m)
    movel([0.115300, -1.331245, -2.563492, -0.817651, 1.570796, 1.686097],accel_mss,speed_ms,0,blend_radius_m)
    movel([0.115300, -1.356498, -2.576059, -0.779832, 1.570796, 1.686097],accel_mss,speed_ms,0,blend_radius_m)
    speed_ms = 0.003
    movel([0.115300, -1.366350, -2.580637, -0.765403, 1.570796, 1.686097],accel_mss,speed_ms,0,blend_radius_m)
    speed_ms = 0.007
    movel([0.115147, -1.366199, -2.580740, -0.765450, 1.570796, 1.685943],accel_mss,speed_ms,0,blend_radius_m)
    movel([0.115161, -1.365756, -2.581044, -0.765589, 1.570796, 1.685958],accel_mss,speed_ms,0,blend_radius_m)
    movel([0.114937, -1.365561, -2.581178, -0.765651, 1.570796, 1.685734],accel_mss,speed_ms,0,blend_radius_m)
    movel([0.114685, -1.365743, -2.581052, -0.765593, 1.570796, 1.685482],accel_mss,speed_ms,0,blend_radius_m)
    movel([0.114564, -1.365999, -2.580877, -0.765513, 1.570796, 1.685360],accel_mss,speed_ms,0,blend_radius_m)
    movel([0.114505, -1.366260, -2.580699, -0.765431, 1.570796, 1.685301],accel_mss,speed_ms,0,blend_radius_m)
    movel([0.114305, -1.366479, -2.580548, -0.765362, 1.570796, 1.685101],accel_mss,speed_ms,0,blend_radius_m)
    movel([0.114150, -1.366331, -2.580649, -0.765408, 1.570796, 1.684947],accel_mss,speed_ms,0,blend_radius_m)
    movel([0.114152, -1.365911, -2.580937, -0.765540, 1.570796, 1.684948],accel_mss,speed_ms,0,blend_radius_m)
    movel([0.114050, -1.365717, -2.581071, -0.765602, 1.570796, 1.684846],accel_mss,speed_ms,0,blend_radius_m)
    movel([0.113872, -1.365616, -2.581140, -0.765634, 1.570796, 1.684668],accel_mss,speed_ms,0,blend_radius_m)
    movel([0.113440, -1.365643, -2.581121, -0.765625, 1.570796, 1.684236],accel_mss,speed_ms,0,blend_radius_m)
    movel([0.113058, -1.365470, -2.581240, -0.765680, 1.570796, 1.683854],accel_mss,speed_ms,0,blend_radius_m)
    movel([0.112877, -1.365278, -2.581371, -0.765740, 1.570796, 1.683673],accel_mss,speed_ms,0,blend_radius_m)
    movel([0.112754, -1.365018, -2.581549, -0.765822, 1.570796, 1.683550],accel_mss,speed_ms,0,blend_radius_m)
    movel([0.112941, -1.364690, -2.581773, -0.765926, 1.570796, 1.683737],accel_mss,speed_ms,0,blend_radius_m)
    movel([0.113216, -1.364401, -2.581970, -0.766017, 1.570796, 1.684013],accel_mss,speed_ms,0,blend_radius_m)
    movel([0.113587, -1.364309, -2.582033, -0.766047, 1.570796, 1.684383],accel_mss,speed_ms,0,blend_radius_m)
    movel([0.113919, -1.364304, -2.582037, -0.766048, 1.570796, 1.684715],accel_mss,speed_ms,0,blend_radius_m)
    movel([0.114137, -1.364361, -2.581997, -0.766030, 1.570796, 1.684933],accel_mss,speed_ms,0,blend_radius_m)
    movel([0.114307, -1.364503, -2.581901, -0.765985, 1.570796, 1.685103],accel_mss,speed_ms,0,blend_radius_m)
    movel([0.114482, -1.364779, -2.581712, -0.765898, 1.570796, 1.685278],accel_mss,speed_ms,0,blend_radius_m)
    movel([0.114658, -1.365037, -2.581536, -0.765816, 1.570796, 1.685455],accel_mss,speed_ms,0,blend_radius_m)
    movel([0.114837, -1.365132, -2.581471, -0.765786, 1.570796, 1.685633],accel_mss,speed_ms,0,blend_radius_m)
    movel([0.115325, -1.364910, -2.581623, -0.765856, 1.570796, 1.686121],accel_mss,speed_ms,0,blend_radius_m)
    movel([0.115621, -1.364725, -2.581749, -0.765915, 1.570796, 1.686417],accel_mss,speed_ms,0,blend_radius_m)
    movel([0.115907, -1.364643, -2.581805, -0.765941, 1.570796, 1.686703],accel_mss,speed_ms,0,blend_radius_m)
    movel([0.116371, -1.364357, -2.582001, -0.766032, 1.570796, 1.687167],accel_mss,speed_ms,0,blend_radius_m)
    movel([0.116464, -1.364121, -2.582162, -0.766106, 1.570796, 1.687260],accel_mss,speed_ms,0,blend_radius_m)
    movel([0.116312, -1.363881, -2.582325, -0.766182, 1.570796, 1.687108],accel_mss,speed_ms,0,blend_radius_m)
    movel([0.116012, -1.364107, -2.582171, -0.766111, 1.570796, 1.686808],accel_mss,speed_ms,0,blend_radius_m)
    movel([0.115646, -1.364425, -2.581954, -0.766010, 1.570796, 1.686443],accel_mss,speed_ms,0,blend_radius_m)
    movel([0.115581, -1.364176, -2.582124, -0.766089, 1.570796, 1.686377],accel_mss,speed_ms,0,blend_radius_m)
    movel([0.115831, -1.363884, -2.582323, -0.766181, 1.570796, 1.686627],accel_mss,speed_ms,0,blend_radius_m)
    movel([0.116106, -1.363605, -2.582514, -0.766270, 1.570796, 1.686902],accel_mss,speed_ms,0,blend_radius_m)
    movel([0.116442, -1.363532, -2.582564, -0.766294, 1.570796, 1.687238],accel_mss,speed_ms,0,blend_radius_m)
    movel([0.116664, -1.363637, -2.582492, -0.766260, 1.570796, 1.687460],accel_mss,speed_ms,0,blend_radius_m)
    movel([0.116856, -1.363863, -2.582338, -0.766188, 1.570796, 1.687653],accel_mss,speed_ms,0,blend_radius_m)
    movel([0.116823, -1.364149, -2.582142, -0.766097, 1.570796, 1.687619],accel_mss,speed_ms,0,blend_radius_m)
    movel([0.116538, -1.364541, -2.581875, -0.765973, 1.570796, 1.687334],accel_mss,speed_ms,0,blend_radius_m)
    movel([0.115912, -1.365137, -2.581468, -0.765785, 1.570796, 1.686708],accel_mss,speed_ms,0,blend_radius_m)
    movel([0.115665, -1.365447, -2.581255, -0.765687, 1.570796, 1.686461],accel_mss,speed_ms,0,blend_radius_m)
    movel([0.115550, -1.365853, -2.580977, -0.765559, 1.570796, 1.686346],accel_mss,speed_ms,0,blend_radius_m)
    movel([0.115461, -1.366207, -2.580735, -0.765447, 1.570796, 1.686258],accel_mss,speed_ms,0,blend_radius_m)
    speed_ms = 0.003
    movel([0.115300, -1.369680, -2.582146, -0.760563, 1.570796, 1.686097],accel_mss,speed_ms,0,blend_radius_m)
    speed_ms = 0.007
    movel([0.115147, -1.369530, -2.582249, -0.760610, 1.570796, 1.685943],accel_mss,speed_ms,0,blend_radius_m)
    movel([0.115161, -1.369088, -2.582554, -0.760747, 1.570796, 1.685958],accel_mss,speed_ms,0,blend_radius_m)
    movel([0.114937, -1.368893, -2.582688, -0.760808, 1.570796, 1.685734],accel_mss,speed_ms,0,blend_radius_m)
    movel([0.114685, -1.369075, -2.582562, -0.760751, 1.570796, 1.685482],accel_mss,speed_ms,0,blend_radius_m)
    movel([0.114564, -1.369331, -2.582387, -0.760671, 1.570796, 1.685360],accel_mss,speed_ms,0,blend_radius_m)
    movel([0.114505, -1.369590, -2.582208, -0.760591, 1.570796, 1.685301],accel_mss,speed_ms,0,blend_radius_m)
    movel([0.114305, -1.369810, -2.582057, -0.760523, 1.570796, 1.685101],accel_mss,speed_ms,0,blend_radius_m)
    movel([0.114150, -1.369662, -2.582158, -0.760569, 1.570796, 1.684947],accel_mss,speed_ms,0,blend_radius_m)
    movel([0.114152, -1.369243, -2.582447, -0.760699, 1.570796, 1.684948],accel_mss,speed_ms,0,blend_radius_m)
    movel([0.114050, -1.369049, -2.582581, -0.760759, 1.570796, 1.684846],accel_mss,speed_ms,0,blend_radius_m)
    movel([0.113872, -1.368948, -2.582650, -0.760791, 1.570796, 1.684668],accel_mss,speed_ms,0,blend_radius_m)
    movel([0.113440, -1.368975, -2.582631, -0.760782, 1.570796, 1.684236],accel_mss,speed_ms,0,blend_radius_m)
    movel([0.113058, -1.368803, -2.582750, -0.760836, 1.570796, 1.683854],accel_mss,speed_ms,0,blend_radius_m)
    movel([0.112877, -1.368611, -2.582882, -0.760896, 1.570796, 1.683673],accel_mss,speed_ms,0,blend_radius_m)
    movel([0.112754, -1.368352, -2.583060, -0.760977, 1.570796, 1.683550],accel_mss,speed_ms,0,blend_radius_m)
    movel([0.112941, -1.368025, -2.583285, -0.761079, 1.570796, 1.683737],accel_mss,speed_ms,0,blend_radius_m)
    movel([0.113216, -1.367737, -2.583483, -0.761169, 1.570796, 1.684013],accel_mss,speed_ms,0,blend_radius_m)
    movel([0.113587, -1.367646, -2.583545, -0.761198, 1.570796, 1.684383],accel_mss,speed_ms,0,blend_radius_m)
    movel([0.113919, -1.367640, -2.583549, -0.761200, 1.570796, 1.684715],accel_mss,speed_ms,0,blend_radius_m)
    movel([0.114137, -1.367697, -2.583510, -0.761182, 1.570796, 1.684933],accel_mss,speed_ms,0,blend_radius_m)
    movel([0.114307, -1.367839, -2.583413, -0.761137, 1.570796, 1.685103],accel_mss,speed_ms,0,blend_radius_m)
    movel([0.114482, -1.368114, -2.583224, -0.761051, 1.570796, 1.685278],accel_mss,speed_ms,0,blend_radius_m)
    movel([0.114658, -1.368371, -2.583047, -0.760971, 1.570796, 1.685455],accel_mss,speed_ms,0,blend_radius_m)
    movel([0.114837, -1.368465, -2.582982, -0.760941, 1.570796, 1.685633],accel_mss,speed_ms,0,blend_radius_m)
    movel([0.115325, -1.368244, -2.583134, -0.761011, 1.570796, 1.686121],accel_mss,speed_ms,0,blend_radius_m)
    movel([0.115621, -1.368060, -2.583261, -0.761068, 1.570796, 1.686417],accel_mss,speed_ms,0,blend_radius_m)
    movel([0.115907, -1.367978, -2.583317, -0.761094, 1.570796, 1.686703],accel_mss,speed_ms,0,blend_radius_m)
    movel([0.116371, -1.367693, -2.583513, -0.761183, 1.570796, 1.687167],accel_mss,speed_ms,0,blend_radius_m)
    movel([0.116464, -1.367457, -2.583675, -0.761257, 1.570796, 1.687260],accel_mss,speed_ms,0,blend_radius_m)
    movel([0.116312, -1.367218, -2.583838, -0.761332, 1.570796, 1.687108],accel_mss,speed_ms,0,blend_radius_m)
    movel([0.116012, -1.367444, -2.583684, -0.761261, 1.570796, 1.686808],accel_mss,speed_ms,0,blend_radius_m)
    movel([0.115646, -1.367760, -2.583467, -0.761162, 1.570796, 1.686443],accel_mss,speed_ms,0,blend_radius_m)
    movel([0.115581, -1.367513, -2.583637, -0.761240, 1.570796, 1.686377],accel_mss,speed_ms,0,blend_radius_m)
    movel([0.115831, -1.367222, -2.583836, -0.761331, 1.570796, 1.686627],accel_mss,speed_ms,0,blend_radius_m)
    movel([0.116106, -1.366943, -2.584028, -0.761419, 1.570796, 1.686902],accel_mss,speed_ms,0,blend_radius_m)
    movel([0.116442, -1.366870, -2.584077, -0.761442, 1.570796, 1.687238],accel_mss,speed_ms,0,blend_radius_m)
    movel([0.116664, -1.366974, -2.584006, -0.761409, 1.570796, 1.687460],accel_mss,speed_ms,0,blend_radius_m)
    movel([0.116856, -1.367200, -2.583851, -0.761338, 1.570796, 1.687653],accel_mss,speed_ms,0,blend_radius_m)
    movel([0.116823, -1.367486, -2.583655, -0.761248, 1.570796, 1.687619],accel_mss,speed_ms,0,blend_radius_m)
    movel([0.116538, -1.367876, -2.583387, -0.761126, 1.570796, 1.687334],accel_mss,speed_ms,0,blend_radius_m)
    movel([0.115912, -1.368471, -2.582979, -0.760940, 1.570796, 1.686708],accel_mss,speed_ms,0,blend_radius_m)
    movel([0.115665, -1.368780, -2.582766, -0.760843, 1.570796, 1.686461],accel_mss,speed_ms,0,blend_radius_m)
    movel([0.115550, -1.369185, -2.582487, -0.760717, 1.570796, 1.686346],accel_mss,speed_ms,0,blend_radius_m)
    movel([0.115461, -1.369538, -2.582244, -0.760607, 1.570796, 1.686258],accel_mss,speed_ms,0,blend_radius_m)
    speed_ms = 0.003
    movel([0.115300, -1.356498, -2.576059, -0.779832, 1.570796, 1.686097],accel_mss,speed_ms,0,blend_radius_m)
    speed_ms = 1.000
    movel([0.115300, -1.331245, -2.563492, -0.817651, 1.570796, 1.686097],accel_mss,speed_ms,0,blend_radius_m)
    movel([0.114036, -1.330032, -2.564282, -0.818075, 1.570796, 1.684833],accel_mss,speed_ms,0,blend_radius_m)
    movel([0.114036, -1.355305, -2.576864, -0.780220, 1.570796, 1.684833],accel_mss,speed_ms,0,blend_radius_m)
    speed_ms = 0.003
    movel([0.114036, -1.365165, -2.581448, -0.765776, 1.570796, 1.684833],accel_mss,speed_ms,0,blend_radius_m)
    speed_ms = 0.007
    movel([0.113723, -1.365329, -2.581336, -0.765724, 1.570796, 1.684520],accel_mss,speed_ms,0,blend_radius_m)
    movel([0.113357, -1.365280, -2.581370, -0.765739, 1.570796, 1.684153],accel_mss,speed_ms,0,blend_radius_m)
    movel([0.113127, -1.365067, -2.581515, -0.765807, 1.570796, 1.683924],accel_mss,speed_ms,0,blend_radius_m)
    movel([0.113178, -1.364791, -2.581704, -0.765894, 1.570796, 1.683974],accel_mss,speed_ms,0,blend_radius_m)
    movel([0.113608, -1.364574, -2.581852, -0.765963, 1.570796, 1.684405],accel_mss,speed_ms,0,blend_radius_m)
    movel([0.113870, -1.364583, -2.581846, -0.765960, 1.570796, 1.684666],accel_mss,speed_ms,0,blend_radius_m)
    movel([0.114043, -1.364683, -2.581778, -0.765928, 1.570796, 1.684839],accel_mss,speed_ms,0,blend_radius_m)
    movel([0.114163, -1.364837, -2.581673, -0.765879, 1.570796, 1.684959],accel_mss,speed_ms,0,blend_radius_m)
    movel([0.114036, -1.365165, -2.581448, -0.765776, 1.570796, 1.684833],accel_mss,speed_ms,0,blend_radius_m)
    speed_ms = 0.003
    movel([0.114036, -1.368499, -2.582959, -0.760931, 1.570796, 1.684833],accel_mss,speed_ms,0,blend_radius_m)
    speed_ms = 0.007
    movel([0.113723, -1.368662, -2.582847, -0.760880, 1.570796, 1.684520],accel_mss,speed_ms,0,blend_radius_m)
    movel([0.113357, -1.368613, -2.582880, -0.760895, 1.570796, 1.684153],accel_mss,speed_ms,0,blend_radius_m)
    movel([0.113127, -1.368401, -2.583026, -0.760962, 1.570796, 1.683924],accel_mss,speed_ms,0,blend_radius_m)
    movel([0.113178, -1.368126, -2.583215, -0.761047, 1.570796, 1.683974],accel_mss,speed_ms,0,blend_radius_m)
    movel([0.113608, -1.367909, -2.583364, -0.761115, 1.570796, 1.684405],accel_mss,speed_ms,0,blend_radius_m)
    movel([0.113870, -1.367919, -2.583358, -0.761112, 1.570796, 1.684666],accel_mss,speed_ms,0,blend_radius_m)
    movel([0.114043, -1.368018, -2.583289, -0.761081, 1.570796, 1.684839],accel_mss,speed_ms,0,blend_radius_m)
    movel([0.114163, -1.368172, -2.583184, -0.761033, 1.570796, 1.684959],accel_mss,speed_ms,0,blend_radius_m)
    movel([0.114036, -1.368499, -2.582959, -0.760931, 1.570796, 1.684833],accel_mss,speed_ms,0,blend_radius_m)
    speed_ms = 0.003
    movel([0.114036, -1.355305, -2.576864, -0.780220, 1.570796, 1.684833],accel_mss,speed_ms,0,blend_radius_m)
    speed_ms = 1.000
    movel([0.114036, -1.330032, -2.564282, -0.818075, 1.570796, 1.684833],accel_mss,speed_ms,0,blend_radius_m)
    movel([0.107334, -1.332493, -2.562679, -0.817217, 1.570796, 1.678130],accel_mss,speed_ms,0,blend_radius_m)
    movel([0.107334, -1.357724, -2.575230, -0.779436, 1.570796, 1.678130],accel_mss,speed_ms,0,blend_radius_m)
    speed_ms = 0.003
    movel([0.107334, -1.367566, -2.579801, -0.765021, 1.570796, 1.678130],accel_mss,speed_ms,0,blend_radius_m)
    speed_ms = 0.007
    movel([0.107250, -1.368281, -2.579310, -0.764798, 1.570796, 1.678047],accel_mss,speed_ms,0,blend_radius_m)
    movel([0.107024, -1.368666, -2.579044, -0.764679, 1.570796, 1.677820],accel_mss,speed_ms,0,blend_radius_m)
    movel([0.106591, -1.369021, -2.578799, -0.764568, 1.570796, 1.677388],accel_mss,speed_ms,0,blend_radius_m)
    movel([0.105893, -1.369496, -2.578472, -0.764421, 1.570796, 1.676689],accel_mss,speed_ms,0,blend_radius_m)
    movel([0.105181, -1.369942, -2.578164, -0.764283, 1.570796, 1.675977],accel_mss,speed_ms,0,blend_radius_m)
    movel([0.104870, -1.369983, -2.578136, -0.764270, 1.570796, 1.675666],accel_mss,speed_ms,0,blend_radius_m)
    movel([0.104761, -1.369797, -2.578264, -0.764328, 1.570796, 1.675557],accel_mss,speed_ms,0,blend_radius_m)
    movel([0.104653, -1.368422, -2.579213, -0.764755, 1.570796, 1.675449],accel_mss,speed_ms,0,blend_radius_m)
